LIN {X 0,Y 359.815,Z 382.386,A -85,B 0,C 180,E1 -13821.382,E2 -13821.382} C_VEL
LIN {X 0,Y 358.544,Z 382.558,A -85,B 0,C 180,E1 -13823.982,E2 -13823.982} C_VEL
LIN {X 0,Y 356.991,Z 383.681,A -85,B 0,C 180,E1 -13826.549,E2 -13826.549} C_VEL
LIN {X 0,Y 355.028,Z 386.583,A -85,B 0,C 180,E1 -13830.579,E2 -13830.579} C_VEL
LIN {X 0,Y 354.271,Z 388.561,A -85,B 0,C 180,E1 -13832.654,E2 -13832.654} C_VEL
LIN {X 0,Y 355.693,Z 391.608,A -85,B 0,C 180,E1 -13833.25,E2 -13833.25} C_VEL
LIN {X 0,Y 359.376,Z 398.785,A -85,B 0,C 180,E1 -13834.634,E2 -13834.634} C_VEL
LIN {X 0,Y 363.625,Z 409.562,A -85,B 0,C 180,E1 -13836.413,E2 -13836.413} C_VEL
LIN {X 0,Y 366.259,Z 418.959,A -85,B 0,C 180,E1 -13837.81,E2 -13837.81} C_VEL
LIN {X 0,Y 364.007,Z 432.05,A -85,B 0,C 180,E1 -13839.073,E2 -13839.073} C_VEL
LIN {X 0,Y 361.656,Z 444.882,A -85,B 0,C 180,E1 -13840.562,E2 -13840.562} C_VEL
LIN {X 0,Y 359.281,Z 457.215,A -85,B 0,C 180,E1 -13842.351,E2 -13842.351} C_VEL
LIN {X 0,Y 357.338,Z 466.693,A -85,B 0,C 180,E1 -13844.018,E2 -13844.018} C_VEL
LIN {X 0,Y 355.42,Z 475.697,A -85,B 0,C 180,E1 -13845.971,E2 -13845.971} C_VEL
LIN {X 0,Y 353.712,Z 483.022,A -85,B 0,C 180,E1 -13847.959,E2 -13847.959} C_VEL
LIN {X 0,Y 352.415,Z 488.041,A -85,B 0,C 180,E1 -13849.661,E2 -13849.661} C_VEL
LIN {X 0,Y 351.389,Z 491.946,A -85,B 0,C 180,E1 -13851.373,E2 -13851.373} C_VEL
LIN {X 0,Y 350.548,Z 494.863,A -85,B 0,C 180,E1 -13853.092,E2 -13853.092} C_VEL
LIN {X 0,Y 350.216,Z 496.262,A -85,B 0,C 180,E1 -13854.242,E2 -13854.242} C_VEL
LIN {X 0,Y 349.782,Z 497.289,A -85,B 0,C 180,E1 -13855.391,E2 -13855.391} C_VEL
LIN {X 0,Y 349.427,Z 497.902,A -85,B 0,C 180,E1 -13856.541,E2 -13856.541} C_VEL
LIN {X 0,Y 349.043,Z 498.099,A -85,B 0,C 180,E1 -13857.693,E2 -13857.693} C_VEL
LIN {X 0,Y 348.804,Z 497.883,A -85,B 0,C 180,E1 -13858.846,E2 -13858.846} C_VEL
LIN {X 0,Y 348.65,Z 497.262,A -85,B 0,C 180,E1 -13860,E2 -13860} C_VEL
LIN {X 0,Y 348.523,Z 496.239,A -85,B 0,C 180,E1 -13861.156,E2 -13861.156} C_VEL
LIN {X 0,Y 348.44,Z 494.801,A -85,B 0,C 180,E1 -13862.312,E2 -13862.312} C_VEL
LIN {X 0,Y 348.542,Z 491.806,A -85,B 0,C 180,E1 -13864.047,E2 -13864.047} C_VEL
LIN {X 0,Y 348.425,Z 487.85,A -85,B 0,C 180,E1 -13865.789,E2 -13865.789} C_VEL
LIN {X 0,Y 348.951,Z 482.756,A -85,B 0,C 180,E1 -13867.523,E2 -13867.523} C_VEL
LIN {X 0,Y 349.426,Z 475.921,A -85,B 0,C 180,E1 -13869.414,E2 -13869.414} C_VEL
LIN {X 0,Y 349.993,Z 467.529,A -85,B 0,C 180,E1 -13871.291,E2 -13871.291} C_VEL
LIN {X 0,Y 350.742,Z 458.089,A -85,B 0,C 180,E1 -13873.028,E2 -13873.028} C_VEL
LIN {X 0,Y 351.6,Z 447.694,A -85,B 0,C 180,E1 -13874.617,E2 -13874.617} C_VEL
LIN {X 0,Y 352.616,Z 435.041,A -85,B 0,C 180,E1 -13876.203,E2 -13876.203} C_VEL
LIN {X 0,Y 353.463,Z 422.474,A -85,B 0,C 180,E1 -13877.502,E2 -13877.502} C_VEL
LIN {X 0,Y 354.563,Z 408.916,A -85,B 0,C 180,E1 -13878.616,E2 -13878.616} C_VEL
LIN {X 0,Y 354.923,Z 402.075,A -85,B 0,C 180,E1 -13879.097,E2 -13879.097} C_VEL
LIN {X 0,Y 353.011,Z 392.134,A -85,B 0,C 180,E1 -13879.828,E2 -13879.828} C_VEL
LIN {X 0,Y 349.184,Z 376.619,A -85,B 0,C 180,E1 -13880.804,E2 -13880.804} C_VEL
LIN {X 0,Y 347.875,Z 371.28,A -85,B 0,C 180,E1 -13881.095,E2 -13881.095} C_VEL
LIN {X 0,Y 348.164,Z 364.382,A -85,B 0,C 180,E1 -13885.082,E2 -13885.082} C_VEL
LIN {X 0,Y 348.529,Z 357.832,A -85,B 0,C 180,E1 -13888.944,E2 -13888.944} C_VEL
LIN {X 0,Y 348.812,Z 352.473,A -85,B 0,C 180,E1 -13892.192,E2 -13892.192} C_VEL
LIN {X 0,Y 349.02,Z 347.907,A -85,B 0,C 180,E1 -13895.022,E2 -13895.022} C_VEL
LIN {X 0,Y 348.92,Z 344.539,A -85,B 0,C 180,E1 -13897.177,E2 -13897.177} C_VEL
LIN {X 0,Y 348.056,Z 338.972,A -85,B 0,C 180,E1 -13900.918,E2 -13900.918} C_VEL
LIN {X 0,Y 347.764,Z 337.48,A -85,B 0,C 180,E1 -13902.023,E2 -13902.023} C_VEL
LIN {X 0,Y 347.739,Z 337.481,A -85,B 0,C 180,E1 -13906.392,E2 -13906.392} C_VEL
LIN {X 0,Y 347.767,Z 337.702,A -85,B 0,C 180,E1 -13906.68,E2 -13906.68} C_VEL
LIN {X 0,Y 349.289,Z 344.678,A -85,B 0,C 180,E1 -13909.917,E2 -13909.917} C_VEL
LIN {X 0,Y 350.445,Z 351.066,A -85,B 0,C 180,E1 -13913.01,E2 -13913.01} C_VEL
LIN {X 0,Y 350.698,Z 355.843,A -85,B 0,C 180,E1 -13915.25,E2 -13915.25} C_VEL
LIN {X 0,Y 350.454,Z 364.261,A -85,B 0,C 180,E1 -13919.175,E2 -13919.175} C_VEL
LIN {X 0,Y 350.383,Z 371.52,A -85,B 0,C 180,E1 -13922.524,E2 -13922.524} C_VEL
LIN {X 0,Y 350.5,Z 380.256,A -85,B 0,C 180,E1 -13926.355,E2 -13926.355} C_VEL
LIN {X 0,Y 350.722,Z 387.896,A -85,B 0,C 180,E1 -13929.358,E2 -13929.358} C_VEL
LIN {X 0,Y 354.939,Z 400.483,A -85,B 0,C 180,E1 -13930.039,E2 -13930.039} C_VEL
LIN {X 0,Y 356.418,Z 406.371,A -85,B 0,C 180,E1 -13930.412,E2 -13930.412} C_VEL
LIN {X 0,Y 355.912,Z 419.475,A -85,B 0,C 180,E1 -13931.193,E2 -13931.193} C_VEL
LIN {X 0,Y 355.256,Z 430.963,A -85,B 0,C 180,E1 -13932.118,E2 -13932.118} C_VEL
LIN {X 0,Y 354.442,Z 440.978,A -85,B 0,C 180,E1 -13933.14,E2 -13933.14} C_VEL
LIN {X 0,Y 353.309,Z 452.163,A -85,B 0,C 180,E1 -13934.568,E2 -13934.568} C_VEL
LIN {X 0,Y 352.501,Z 460.293,A -85,B 0,C 180,E1 -13935.861,E2 -13935.861} C_VEL
LIN {X 0,Y 351.534,Z 467.81,A -85,B 0,C 180,E1 -13937.293,E2 -13937.293} C_VEL
LIN {X 0,Y 350.826,Z 474.233,A -85,B 0,C 180,E1 -13938.793,E2 -13938.793} C_VEL
LIN {X 0,Y 350.022,Z 480.931,A -85,B 0,C 180,E1 -13940.754,E2 -13940.754} C_VEL
LIN {X 0,Y 349.087,Z 485.6,A -85,B 0,C 180,E1 -13942.478,E2 -13942.478} C_VEL
LIN {X 0,Y 348.671,Z 489.123,A -85,B 0,C 180,E1 -13944.213,E2 -13944.213} C_VEL
LIN {X 0,Y 348.589,Z 490.915,A -85,B 0,C 180,E1 -13945.372,E2 -13945.372} C_VEL
LIN {X 0,Y 348.435,Z 492.298,A -85,B 0,C 180,E1 -13946.528,E2 -13946.528} C_VEL
LIN {X 0,Y 348.086,Z 493.891,A -85,B 0,C 180,E1 -13948.84,E2 -13948.84} C_VEL
LIN {X 0,Y 348.041,Z 494.124,A -85,B 0,C 180,E1 -13949.997,E2 -13949.997} C_VEL
LIN {X 0,Y 348.214,Z 493.353,A -85,B 0,C 180,E1 -13952.311,E2 -13952.311} C_VEL
LIN {X 0,Y 348.446,Z 492.394,A -85,B 0,C 180,E1 -13953.466,E2 -13953.466} C_VEL
LIN {X 0,Y 348.63,Z 491.062,A -85,B 0,C 180,E1 -13954.622,E2 -13954.622} C_VEL
LIN {X 0,Y 348.843,Z 488.284,A -85,B 0,C 180,E1 -13956.359,E2 -13956.359} C_VEL
LIN {X 0,Y 349.415,Z 484.462,A -85,B 0,C 180,E1 -13958.091,E2 -13958.091} C_VEL
LIN {X 0,Y 350.209,Z 479.495,A -85,B 0,C 180,E1 -13959.818,E2 -13959.818} C_VEL
LIN {X 0,Y 350.899,Z 473.265,A -85,B 0,C 180,E1 -13961.551,E2 -13961.551} C_VEL
LIN {X 0,Y 351.86,Z 465.488,A -85,B 0,C 180,E1 -13963.276,E2 -13963.276} C_VEL
LIN {X 0,Y 352.854,Z 457.514,A -85,B 0,C 180,E1 -13964.708,E2 -13964.708} C_VEL
LIN {X 0,Y 353.725,Z 448.821,A -85,B 0,C 180,E1 -13965.999,E2 -13965.999} C_VEL
LIN {X 0,Y 354.637,Z 438.034,A -85,B 0,C 180,E1 -13967.29,E2 -13967.29} C_VEL
LIN {X 0,Y 355.523,Z 426.896,A -85,B 0,C 180,E1 -13968.339,E2 -13968.339} C_VEL
LIN {X 0,Y 356.176,Z 415.355,A -85,B 0,C 180,E1 -13969.184,E2 -13969.184} C_VEL
LIN {X 0,Y 356.421,Z 405.632,A -85,B 0,C 180,E1 -13969.731,E2 -13969.731} C_VEL
LIN {X 0,Y 352.601,Z 393.285,A -85,B 0,C 180,E1 -13970.478,E2 -13970.478} C_VEL
LIN {X 0,Y 350.682,Z 387.643,A -85,B 0,C 180,E1 -13970.78,E2 -13970.78} C_VEL
LIN {X 0,Y 350.472,Z 379.042,A -85,B 0,C 180,E1 -13974.269,E2 -13974.269} C_VEL
LIN {X 0,Y 350.383,Z 370.525,A -85,B 0,C 180,E1 -13978.047,E2 -13978.047} C_VEL
LIN {X 0,Y 350.518,Z 363.233,A -85,B 0,C 180,E1 -13981.416,E2 -13981.416} C_VEL
LIN {X 0,Y 350.65,Z 358.63,A -85,B 0,C 180,E1 -13983.61,E2 -13983.61} C_VEL
LIN {X 0,Y 350.02,Z 356.826,A -85,B 0,C 180,E1 -13984.524,E2 -13984.524} C_VEL
LIN {X 0,Y 347.188,Z 354.458,A -85,B 0,C 180,E1 -13986.037,E2 -13986.037} C_VEL
LIN {X 0,Y 344.649,Z 352.626,A -85,B 0,C 180,E1 -13987.263,E2 -13987.263} C_VEL
LIN {X 0,Y 343.379,Z 350.969,A -85,B 0,C 180,E1 -13988.198,E2 -13988.198} C_VEL
LIN {X 0,Y 343.181,Z 350.325,A -85,B 0,C 180,E1 -13988.512,E2 -13988.512} C_VEL
LIN {X 0,Y 342.135,Z 345.025,A -85,B 0,C 180,E1 -13991.092,E2 -13991.092} C_VEL
LIN {X 0,Y 340.707,Z 338.358,A -85,B 0,C 180,E1 -13994.205,E2 -13994.205} C_VEL
LIN {X 0,Y 340.733,Z 338.353,A -85,B 0,C 180,E1 -13997.943,E2 -13997.943} C_VEL
LIN {X 0,Y 340.719,Z 338.355,A -85,B 0,C 180,E1 -14000.25,E2 -14000.25} C_VEL
LIN {X 0,Y 340.695,Z 338.359,A -85,B 0,C 180,E1 -14003.556,E2 -14003.556} C_VEL
LIN {X 0,Y 340.674,Z 338.361,A -85,B 0,C 180,E1 -14006.151,E2 -14006.151} C_VEL
LIN {X 0,Y 340.755,Z 338.345,A -85,B 0,C 180,E1 -14010.33,E2 -14010.33} C_VEL
LIN {X 0,Y 340.784,Z 338.341,A -85,B 0,C 180,E1 -14013.018,E2 -14013.018} C_VEL
LIN {X 0,Y 340.757,Z 338.343,A -85,B 0,C 180,E1 -14016.929,E2 -14016.929} C_VEL
LIN {X 0,Y 340.785,Z 338.341,A -85,B 0,C 180,E1 -14020.733,E2 -14020.733} C_VEL
LIN {X 0,Y 340.765,Z 338.352,A -85,B 0,C 180,E1 -14023.217,E2 -14023.217} C_VEL
LIN {X 0,Y 340.825,Z 338.338,A -85,B 0,C 180,E1 -14026.889,E2 -14026.889} C_VEL
LIN {X 0,Y 340.908,Z 338.321,A -85,B 0,C 180,E1 -14030.507,E2 -14030.507} C_VEL
LIN {X 0,Y 341.052,Z 338.314,A -85,B 0,C 180,E1 -14032.897,E2 -14032.897} C_VEL
LIN {X 0,Y 341.143,Z 338.304,A -85,B 0,C 180,E1 -14037.638,E2 -14037.638} C_VEL
LIN {X 0,Y 341.252,Z 338.281,A -85,B 0,C 180,E1 -14040,E2 -14040} C_VEL
LIN {X 0,Y 341.157,Z 338.298,A -85,B 0,C 180,E1 -14042.361,E2 -14042.361} C_VEL
LIN {X 0,Y 341.055,Z 338.313,A -85,B 0,C 180,E1 -14047.102,E2 -14047.102} C_VEL
LIN {X 0,Y 340.852,Z 338.341,A -85,B 0,C 180,E1 -14050.694,E2 -14050.694} C_VEL
LIN {X 0,Y 340.839,Z 338.344,A -85,B 0,C 180,E1 -14054.325,E2 -14054.325} C_VEL
LIN {X 0,Y 340.816,Z 338.344,A -85,B 0,C 180,E1 -14058.468,E2 -14058.468} C_VEL
LIN {X 0,Y 340.79,Z 338.346,A -85,B 0,C 180,E1 -14061.883,E2 -14061.883} C_VEL
LIN {X 0,Y 340.754,Z 338.351,A -85,B 0,C 180,E1 -14065.665,E2 -14065.665} C_VEL
LIN {X 0,Y 340.718,Z 338.356,A -85,B 0,C 180,E1 -14068.321,E2 -14068.321} C_VEL
LIN {X 0,Y 340.683,Z 338.371,A -85,B 0,C 180,E1 -14071.132,E2 -14071.132} C_VEL
LIN {X 0,Y 343.277,Z 347.352,A -85,B 0,C 180,E1 -14075.029,E2 -14075.029} C_VEL
LIN {X 0,Y 346.144,Z 357.402,A -85,B 0,C 180,E1 -14079.006,E2 -14079.006} C_VEL
LIN {X 0,Y 348.807,Z 366.887,A -85,B 0,C 180,E1 -14082.452,E2 -14082.452} C_VEL
LIN {X 0,Y 351.893,Z 377.324,A -85,B 0,C 180,E1 -14085.971,E2 -14085.971} C_VEL
LIN {X 0,Y 354.639,Z 387.6,A -85,B 0,C 180,E1 -14089.163,E2 -14089.163} C_VEL
LIN {X 0,Y 355.6,Z 391.91,A -85,B 0,C 180,E1 -14090.424,E2 -14090.424} C_VEL
LIN {X 0,Y 352.415,Z 406.455,A -85,B 0,C 180,E1 -14093.968,E2 -14093.968} C_VEL
LIN {X 0,Y 350.81,Z 414.741,A -85,B 0,C 180,E1 -14095.931,E2 -14095.931} C_VEL
LIN {X 0,Y 354.593,Z 437.489,A -85,B 0,C 180,E1 -14096.931,E2 -14096.931} C_VEL
LIN {X 0,Y 356.863,Z 453.689,A -85,B 0,C 180,E1 -14097.821,E2 -14097.821} C_VEL
LIN {X 0,Y 358.237,Z 464.384,A -85,B 0,C 180,E1 -14098.523,E2 -14098.523} C_VEL
LIN {X 0,Y 356.534,Z 480.109,A -85,B 0,C 180,E1 -14099.501,E2 -14099.501} C_VEL
LIN {X 0,Y 354.425,Z 495.314,A -85,B 0,C 180,E1 -14100.673,E2 -14100.673} C_VEL
LIN {X 0,Y 352.288,Z 509.765,A -85,B 0,C 180,E1 -14102.046,E2 -14102.046} C_VEL
LIN {X 0,Y 349.976,Z 523.578,A -85,B 0,C 180,E1 -14103.625,E2 -14103.625} C_VEL
LIN {X 0,Y 347.716,Z 536.833,A -85,B 0,C 180,E1 -14105.44,E2 -14105.44} C_VEL
LIN {X 0,Y 345.769,Z 548.209,A -85,B 0,C 180,E1 -14107.286,E2 -14107.286} C_VEL
LIN {X 0,Y 343.953,Z 559.081,A -85,B 0,C 180,E1 -14109.365,E2 -14109.365} C_VEL
LIN {X 0,Y 342.497,Z 568.353,A -85,B 0,C 180,E1 -14111.458,E2 -14111.458} C_VEL
LIN {X 0,Y 341.455,Z 576.22,A -85,B 0,C 180,E1 -14113.563,E2 -14113.563} C_VEL
LIN {X 0,Y 340.56,Z 583.613,A -85,B 0,C 180,E1 -14115.91,E2 -14115.91} C_VEL
LIN {X 0,Y 340.047,Z 589.25,A -85,B 0,C 180,E1 -14118.076,E2 -14118.076} C_VEL
LIN {X 0,Y 339.712,Z 594.263,A -85,B 0,C 180,E1 -14120.477,E2 -14120.477} C_VEL
LIN {X 0,Y 339.718,Z 598.574,A -85,B 0,C 180,E1 -14123.219,E2 -14123.219} C_VEL
LIN {X 0,Y 339.696,Z 600.784,A -85,B 0,C 180,E1 -14125.256,E2 -14125.256} C_VEL
LIN {X 0,Y 339.807,Z 601.705,A -85,B 0,C 180,E1 -14126.446,E2 -14126.446} C_VEL
LIN {X 0,Y 339.722,Z 602.725,A -85,B 0,C 180,E1 -14128.818,E2 -14128.818} C_VEL
LIN {X 0,Y 339.738,Z 602.594,A -85,B 0,C 180,E1 -14131.188,E2 -14131.188} C_VEL
LIN {X 0,Y 339.818,Z 601.433,A -85,B 0,C 180,E1 -14133.56,E2 -14133.56} C_VEL
LIN {X 0,Y 339.688,Z 599.113,A -85,B 0,C 180,E1 -14135.941,E2 -14135.941} C_VEL
LIN {X 0,Y 339.756,Z 595.701,A -85,B 0,C 180,E1 -14138.328,E2 -14138.328} C_VEL
LIN {X 0,Y 339.864,Z 591.152,A -85,B 0,C 180,E1 -14140.729,E2 -14140.729} C_VEL
LIN {X 0,Y 340.473,Z 584.037,A -85,B 0,C 180,E1 -14143.629,E2 -14143.629} C_VEL
LIN {X 0,Y 341.443,Z 575.329,A -85,B 0,C 180,E1 -14146.443,E2 -14146.443} C_VEL
LIN {X 0,Y 342.697,Z 566.272,A -85,B 0,C 180,E1 -14148.847,E2 -14148.847} C_VEL
LIN {X 0,Y 344.387,Z 555.599,A -85,B 0,C 180,E1 -14151.24,E2 -14151.24} C_VEL
LIN {X 0,Y 346.328,Z 544.712,A -85,B 0,C 180,E1 -14153.313,E2 -14153.313} C_VEL
LIN {X 0,Y 348.731,Z 532.099,A -85,B 0,C 180,E1 -14155.359,E2 -14155.359} C_VEL
LIN {X 0,Y 351.045,Z 519.623,A -85,B 0,C 180,E1 -14157.097,E2 -14157.097} C_VEL
LIN {X 0,Y 353.86,Z 504.528,A -85,B 0,C 180,E1 -14158.865,E2 -14158.865} C_VEL
LIN {X 0,Y 356.57,Z 489.422,A -85,B 0,C 180,E1 -14160.338,E2 -14160.338} C_VEL
LIN {X 0,Y 359.444,Z 472.332,A -85,B 0,C 180,E1 -14161.702,E2 -14161.702} C_VEL
LIN {X 0,Y 360.438,Z 465.571,A -85,B 0,C 180,E1 -14162.165,E2 -14162.165} C_VEL
LIN {X 0,Y 359.822,Z 450.974,A -85,B 0,C 180,E1 -14163.354,E2 -14163.354} C_VEL
LIN {X 0,Y 359.195,Z 436.999,A -85,B 0,C 180,E1 -14164.365,E2 -14164.365} C_VEL
LIN {X 0,Y 357.293,Z 423.761,A -85,B 0,C 180,E1 -14165.394,E2 -14165.394} C_VEL
LIN {X 0,Y 354.236,Z 409.339,A -85,B 0,C 180,E1 -14166.695,E2 -14166.695} C_VEL
LIN {X 0,Y 357.67,Z 399.95,A -85,B 0,C 180,E1 -14169.551,E2 -14169.551} C_VEL
LIN {X 0,Y 358.302,Z 397.75,A -85,B 0,C 180,E1 -14170.34,E2 -14170.34} C_VEL
LIN {X 0,Y 357.264,Z 393.411,A -85,B 0,C 180,E1 -14172.593,E2 -14172.593} C_VEL
LIN {X 0,Y 355.864,Z 389.527,A -85,B 0,C 180,E1 -14175.316,E2 -14175.316} C_VEL
LIN {X 0,Y 354.871,Z 387.187,A -85,B 0,C 180,E1 -14177.675,E2 -14177.675} C_VEL
LIN {X 0,Y 354.314,Z 386.23,A -85,B 0,C 180,E1 -14179.113,E2 -14179.113} C_VEL
LIN {X 0,Y 353.604,Z 385.549,A -85,B 0,C 180,E1 -14180.82,E2 -14180.82} C_VEL
LIN {X 0,Y 352.494,Z 385.363,A -85,B 0,C 180,E1 -14183.264,E2 -14183.264} C_VEL
LIN {X 0,Y 350.838,Z 386.228,A -85,B 0,C 180,E1 -14185.883,E2 -14185.883} C_VEL
LIN {X 0,Y 348.767,Z 388.633,A -85,B 0,C 180,E1 -14189.75,E2 -14189.75} C_VEL
LIN {X 0,Y 348.145,Z 389.961,A -85,B 0,C 180,E1 -14191.312,E2 -14191.312} C_VEL
LIN {X 0,Y 349.86,Z 393.47,A -85,B 0,C 180,E1 -14192.117,E2 -14192.117} C_VEL
LIN {X 0,Y 353.24,Z 400.153,A -85,B 0,C 180,E1 -14193.552,E2 -14193.552} C_VEL
LIN {X 0,Y 356.955,Z 409.105,A -85,B 0,C 180,E1 -14195.215,E2 -14195.215} C_VEL
LIN {X 0,Y 360.014,Z 419.086,A -85,B 0,C 180,E1 -14196.86,E2 -14196.86} C_VEL
LIN {X 0,Y 360.455,Z 422.118,A -85,B 0,C 180,E1 -14197.294,E2 -14197.294} C_VEL
LIN {X 0,Y 357.903,Z 435.965,A -85,B 0,C 180,E1 -14198.699,E2 -14198.699} C_VEL
LIN {X 0,Y 355.433,Z 448.064,A -85,B 0,C 180,E1 -14200.208,E2 -14200.208} C_VEL
LIN {X 0,Y 353.294,Z 458.324,A -85,B 0,C 180,E1 -14201.742,E2 -14201.742} C_VEL
LIN {X 0,Y 350.898,Z 469.156,A -85,B 0,C 180,E1 -14203.716,E2 -14203.716} C_VEL
LIN {X 0,Y 349.022,Z 477.161,A -85,B 0,C 180,E1 -14205.52,E2 -14205.52} C_VEL
LIN {X 0,Y 347.045,Z 485.046,A -85,B 0,C 180,E1 -14207.724,E2 -14207.724} C_VEL
LIN {X 0,Y 345.673,Z 489.873,A -85,B 0,C 180,E1 -14209.457,E2 -14209.457} C_VEL
LIN {X 0,Y 344.595,Z 493.651,A -85,B 0,C 180,E1 -14211.202,E2 -14211.202} C_VEL
LIN {X 0,Y 343.699,Z 496.45,A -85,B 0,C 180,E1 -14212.953,E2 -14212.953} C_VEL
LIN {X 0,Y 343.32,Z 497.77,A -85,B 0,C 180,E1 -14214.126,E2 -14214.126} C_VEL
LIN {X 0,Y 342.858,Z 498.735,A -85,B 0,C 180,E1 -14215.297,E2 -14215.297} C_VEL
LIN {X 0,Y 342.477,Z 499.268,A -85,B 0,C 180,E1 -14216.471,E2 -14216.471} C_VEL
LIN {X 0,Y 342.091,Z 499.404,A -85,B 0,C 180,E1 -14217.646,E2 -14217.646} C_VEL
LIN {X 0,Y 341.831,Z 499.129,A -85,B 0,C 180,E1 -14218.822,E2 -14218.822} C_VEL
LIN {X 0,Y 341.656,Z 498.447,A -85,B 0,C 180,E1 -14220,E2 -14220} C_VEL
LIN {X 0,Y 341.528,Z 497.365,A -85,B 0,C 180,E1 -14221.18,E2 -14221.18} C_VEL
LIN {X 0,Y 341.434,Z 495.848,A -85,B 0,C 180,E1 -14222.36,E2 -14222.36} C_VEL
LIN {X 0,Y 341.538,Z 492.764,A -85,B 0,C 180,E1 -14224.131,E2 -14224.131} C_VEL
LIN {X 0,Y 341.414,Z 488.707,A -85,B 0,C 180,E1 -14225.908,E2 -14225.908} C_VEL
LIN {X 0,Y 342.068,Z 482.532,A -85,B 0,C 180,E1 -14227.972,E2 -14227.972} C_VEL
LIN {X 0,Y 342.49,Z 475.215,A -85,B 0,C 180,E1 -14229.935,E2 -14229.935} C_VEL
LIN {X 0,Y 343.181,Z 466.57,A -85,B 0,C 180,E1 -14231.818,E2 -14231.818} C_VEL
LIN {X 0,Y 343.922,Z 456.679,A -85,B 0,C 180,E1 -14233.592,E2 -14233.592} C_VEL
LIN {X 0,Y 344.973,Z 445.734,A -85,B 0,C 180,E1 -14235.207,E2 -14235.207} C_VEL
LIN {X 0,Y 345.929,Z 433.274,A -85,B 0,C 180,E1 -14236.737,E2 -14236.737} C_VEL
LIN {X 0,Y 346.796,Z 420.672,A -85,B 0,C 180,E1 -14238.002,E2 -14238.002} C_VEL
LIN {X 0,Y 347.91,Z 407.213,A -85,B 0,C 180,E1 -14239.092,E2 -14239.092} C_VEL
LIN {X 0,Y 348.072,Z 402.371,A -85,B 0,C 180,E1 -14239.436,E2 -14239.436} C_VEL
LIN {X 0,Y 344.914,Z 388.063,A -85,B 0,C 180,E1 -14240.493,E2 -14240.493} C_VEL
LIN {X 0,Y 340.902,Z 371.644,A -85,B 0,C 180,E1 -14241.505,E2 -14241.505} C_VEL
LIN {X 0,Y 341.205,Z 364.583,A -85,B 0,C 180,E1 -14245.63,E2 -14245.63} C_VEL
LIN {X 0,Y 341.531,Z 359.093,A -85,B 0,C 180,E1 -14248.92,E2 -14248.92} C_VEL
LIN {X 0,Y 341.842,Z 353.157,A -85,B 0,C 180,E1 -14252.546,E2 -14252.546} C_VEL
LIN {X 0,Y 342.065,Z 347.941,A -85,B 0,C 180,E1 -14255.843,E2 -14255.843} C_VEL
LIN {X 0,Y 341.649,Z 343.799,A -85,B 0,C 180,E1 -14258.581,E2 -14258.581} C_VEL
LIN {X 0,Y 340.78,Z 338.747,A -85,B 0,C 180,E1 -14262.058,E2 -14262.058} C_VEL
LIN {X 0,Y 340.741,Z 338.352,A -85,B 0,C 180,E1 -14262.419,E2 -14262.419} C_VEL
LIN {X 0,Y 340.7,Z 338.505,A -85,B 0,C 180,E1 -14266.002,E2 -14266.002} C_VEL
LIN {X 0,Y 342.044,Z 344.592,A -85,B 0,C 180,E1 -14268.887,E2 -14268.887} C_VEL
LIN {X 0,Y 343.318,Z 351.214,A -85,B 0,C 180,E1 -14272.109,E2 -14272.109} C_VEL
LIN {X 0,Y 343.879,Z 355.903,A -85,B 0,C 180,E1 -14274.338,E2 -14274.338} C_VEL
LIN {X 0,Y 343.703,Z 363.478,A -85,B 0,C 180,E1 -14277.881,E2 -14277.881} C_VEL
LIN {X 0,Y 343.531,Z 372.203,A -85,B 0,C 180,E1 -14281.928,E2 -14281.928} C_VEL
LIN {X 0,Y 343.621,Z 379.609,A -85,B 0,C 180,E1 -14285.208,E2 -14285.208} C_VEL
LIN {X 0,Y 343.766,Z 387.395,A -85,B 0,C 180,E1 -14288.406,E2 -14288.406} C_VEL
LIN {X 0,Y 343.859,Z 388.871,A -85,B 0,C 180,E1 -14288.925,E2 -14288.925} C_VEL
LIN {X 0,Y 348.143,Z 401.473,A -85,B 0,C 180,E1 -14289.629,E2 -14289.629} C_VEL
LIN {X 0,Y 349.811,Z 408.243,A -85,B 0,C 180,E1 -14290.071,E2 -14290.071} C_VEL
LIN {X 0,Y 349.28,Z 420.787,A -85,B 0,C 180,E1 -14290.84,E2 -14290.84} C_VEL
LIN {X 0,Y 348.583,Z 431.988,A -85,B 0,C 180,E1 -14291.76,E2 -14291.76} C_VEL
LIN {X 0,Y 347.732,Z 442.046,A -85,B 0,C 180,E1 -14292.805,E2 -14292.805} C_VEL
LIN {X 0,Y 346.547,Z 453.235,A -85,B 0,C 180,E1 -14294.259,E2 -14294.259} C_VEL
LIN {X 0,Y 345.7,Z 461.367,A -85,B 0,C 180,E1 -14295.577,E2 -14295.577} C_VEL
LIN {X 0,Y 344.701,Z 468.883,A -85,B 0,C 180,E1 -14297.037,E2 -14297.037} C_VEL
LIN {X 0,Y 343.955,Z 475.257,A -85,B 0,C 180,E1 -14298.552,E2 -14298.552} C_VEL
LIN {X 0,Y 343.104,Z 482.006,A -85,B 0,C 180,E1 -14300.566,E2 -14300.566} C_VEL
LIN {X 0,Y 342.131,Z 486.677,A -85,B 0,C 180,E1 -14302.324,E2 -14302.324} C_VEL
LIN {X 0,Y 341.691,Z 490.2,A -85,B 0,C 180,E1 -14304.094,E2 -14304.094} C_VEL
LIN {X 0,Y 341.611,Z 491.99,A -85,B 0,C 180,E1 -14305.277,E2 -14305.277} C_VEL
LIN {X 0,Y 341.432,Z 493.375,A -85,B 0,C 180,E1 -14306.457,E2 -14306.457} C_VEL
LIN {X 0,Y 341.07,Z 494.968,A -85,B 0,C 180,E1 -14308.816,E2 -14308.816} C_VEL
LIN {X 0,Y 341.046,Z 495.197,A -85,B 0,C 180,E1 -14309.997,E2 -14309.997} C_VEL
LIN {X 0,Y 341.203,Z 494.43,A -85,B 0,C 180,E1 -14312.358,E2 -14312.358} C_VEL
LIN {X 0,Y 341.443,Z 493.47,A -85,B 0,C 180,E1 -14313.537,E2 -14313.537} C_VEL
LIN {X 0,Y 341.645,Z 492.136,A -85,B 0,C 180,E1 -14314.717,E2 -14314.717} C_VEL
LIN {X 0,Y 341.867,Z 489.36,A -85,B 0,C 180,E1 -14316.489,E2 -14316.489} C_VEL
LIN {X 0,Y 342.469,Z 485.536,A -85,B 0,C 180,E1 -14318.256,E2 -14318.256} C_VEL
LIN {X 0,Y 343.301,Z 480.567,A -85,B 0,C 180,E1 -14320.018,E2 -14320.018} C_VEL
LIN {X 0,Y 344.023,Z 474.337,A -85,B 0,C 180,E1 -14321.785,E2 -14321.785} C_VEL
LIN {X 0,Y 345.033,Z 466.558,A -85,B 0,C 180,E1 -14323.544,E2 -14323.544} C_VEL
LIN {X 0,Y 346.069,Z 458.581,A -85,B 0,C 180,E1 -14325.003,E2 -14325.003} C_VEL
LIN {X 0,Y 346.981,Z 449.885,A -85,B 0,C 180,E1 -14326.319,E2 -14326.319} C_VEL
LIN {X 0,Y 347.94,Z 439.091,A -85,B 0,C 180,E1 -14327.634,E2 -14327.634} C_VEL
LIN {X 0,Y 348.88,Z 427.943,A -85,B 0,C 180,E1 -14328.701,E2 -14328.701} C_VEL
LIN {X 0,Y 349.566,Z 415.79,A -85,B 0,C 180,E1 -14329.6,E2 -14329.6} C_VEL
LIN {X 0,Y 349.744,Z 407.09,A -85,B 0,C 180,E1 -14330.101,E2 -14330.101} C_VEL
LIN {X 0,Y 346.163,Z 395.379,A -85,B 0,C 180,E1 -14330.843,E2 -14330.843} C_VEL
LIN {X 0,Y 343.839,Z 388.706,A -85,B 0,C 180,E1 -14331.19,E2 -14331.19} C_VEL
LIN {X 0,Y 343.641,Z 381.411,A -85,B 0,C 180,E1 -14334.14,E2 -14334.14} C_VEL
LIN {X 0,Y 343.568,Z 374.026,A -85,B 0,C 180,E1 -14337.4,E2 -14337.4} C_VEL
LIN {X 0,Y 343.658,Z 366.58,A -85,B 0,C 180,E1 -14340.803,E2 -14340.803} C_VEL
LIN {X 0,Y 343.919,Z 357.864,A -85,B 0,C 180,E1 -14344.898,E2 -14344.898} C_VEL
LIN {X 0,Y 343.616,Z 353.19,A -85,B 0,C 180,E1 -14347.091,E2 -14347.091} C_VEL
LIN {X 0,Y 343.181,Z 350.325,A -85,B 0,C 180,E1 -14348.512,E2 -14348.512} C_VEL
LIN {X 0,Y 342.163,Z 348.602,A -85,B 0,C 180,E1 -14349.439,E2 -14349.439} C_VEL
LIN {X 0,Y 338.792,Z 346.418,A -85,B 0,C 180,E1 -14350.963,E2 -14350.963} C_VEL
LIN {X 0,Y 335.944,Z 344.578,A -85,B 0,C 180,E1 -14352.197,E2 -14352.197} C_VEL
LIN {X 0,Y 334.527,Z 342.849,A -85,B 0,C 180,E1 -14353.144,E2 -14353.144} C_VEL
LIN {X 0,Y 334.299,Z 342.177,A -85,B 0,C 180,E1 -14353.462,E2 -14353.462} C_VEL
LIN {X 0,Y 333.66,Z 339.236,A -85,B 0,C 180,E1 -14354.856,E2 -14354.856} C_VEL
LIN {X 0,Y 333.679,Z 339.232,A -85,B 0,C 180,E1 -14357.624,E2 -14357.624} C_VEL
LIN {X 0,Y 333.668,Z 339.235,A -85,B 0,C 180,E1 -14361.193,E2 -14361.193} C_VEL
LIN {X 0,Y 333.668,Z 339.234,A -85,B 0,C 180,E1 -14365.223,E2 -14365.223} C_VEL
LIN {X 0,Y 333.679,Z 339.228,A -85,B 0,C 180,E1 -14369.635,E2 -14369.635} C_VEL
LIN {X 0,Y 333.723,Z 339.227,A -85,B 0,C 180,E1 -14372.399,E2 -14372.399} C_VEL
LIN {X 0,Y 333.741,Z 339.226,A -85,B 0,C 180,E1 -14375.091,E2 -14375.091} C_VEL
LIN {X 0,Y 333.703,Z 339.23,A -85,B 0,C 180,E1 -14379.02,E2 -14379.02} C_VEL
LIN {X 0,Y 333.774,Z 339.213,A -85,B 0,C 180,E1 -14381.588,E2 -14381.588} C_VEL
LIN {X 0,Y 333.786,Z 339.207,A -85,B 0,C 180,E1 -14385.575,E2 -14385.575} C_VEL
LIN {X 0,Y 333.817,Z 339.213,A -85,B 0,C 180,E1 -14389.077,E2 -14389.077} C_VEL
LIN {X 0,Y 334.002,Z 339.192,A -85,B 0,C 180,E1 -14392.747,E2 -14392.747} C_VEL
LIN {X 0,Y 333.785,Z 339.208,A -85,B 0,C 180,E1 -14395.168,E2 -14395.168} C_VEL
LIN {X 0,Y 334.08,Z 339.184,A -85,B 0,C 180,E1 -14397.588,E2 -14397.588} C_VEL
LIN {X 0,Y 334.204,Z 339.158,A -85,B 0,C 180,E1 -14400,E2 -14400} C_VEL
LIN {X 0,Y 334.119,Z 339.175,A -85,B 0,C 180,E1 -14402.411,E2 -14402.411} C_VEL
LIN {X 0,Y 334.004,Z 339.192,A -85,B 0,C 180,E1 -14407.252,E2 -14407.252} C_VEL
LIN {X 0,Y 333.814,Z 339.217,A -85,B 0,C 180,E1 -14410.922,E2 -14410.922} C_VEL
LIN {X 0,Y 333.785,Z 339.22,A -85,B 0,C 180,E1 -14414.635,E2 -14414.635} C_VEL
LIN {X 0,Y 333.775,Z 339.221,A -85,B 0,C 180,E1 -14418.657,E2 -14418.657} C_VEL
LIN {X 0,Y 333.726,Z 339.227,A -85,B 0,C 180,E1 -14422.275,E2 -14422.275} C_VEL
LIN {X 0,Y 333.715,Z 339.227,A -85,B 0,C 180,E1 -14426.247,E2 -14426.247} C_VEL
LIN {X 0,Y 333.686,Z 339.309,A -85,B 0,C 180,E1 -14430.177,E2 -14430.177} C_VEL
LIN {X 0,Y 336.314,Z 348.652,A -85,B 0,C 180,E1 -14434.348,E2 -14434.348} C_VEL
LIN {X 0,Y 338.865,Z 357.571,A -85,B 0,C 180,E1 -14437.997,E2 -14437.997} C_VEL
LIN {X 0,Y 341.588,Z 367.203,A -85,B 0,C 180,E1 -14441.624,E2 -14441.624} C_VEL
LIN {X 0,Y 344.832,Z 378.406,A -85,B 0,C 180,E1 -14445.506,E2 -14445.506} C_VEL
LIN {X 0,Y 347.626,Z 388.765,A -85,B 0,C 180,E1 -14448.808,E2 -14448.808} C_VEL
LIN {X 0,Y 348.757,Z 393.382,A -85,B 0,C 180,E1 -14450.198,E2 -14450.198} C_VEL
LIN {X 0,Y 345.745,Z 406.685,A -85,B 0,C 180,E1 -14453.523,E2 -14453.523} C_VEL
LIN {X 0,Y 344.169,Z 414.44,A -85,B 0,C 180,E1 -14455.403,E2 -14455.403} C_VEL
LIN {X 0,Y 347.786,Z 437.013,A -85,B 0,C 180,E1 -14456.413,E2 -14456.413} C_VEL
LIN {X 0,Y 350.147,Z 453.357,A -85,B 0,C 180,E1 -14457.338,E2 -14457.338} C_VEL
LIN {X 0,Y 351.555,Z 465.355,A -85,B 0,C 180,E1 -14458.142,E2 -14458.142} C_VEL
LIN {X 0,Y 349.74,Z 481.28,A -85,B 0,C 180,E1 -14459.179,E2 -14459.179} C_VEL
LIN {X 0,Y 347.518,Z 496.549,A -85,B 0,C 180,E1 -14460.412,E2 -14460.412} C_VEL
LIN {X 0,Y 345.406,Z 510.339,A -85,B 0,C 180,E1 -14461.77,E2 -14461.77} C_VEL
LIN {X 0,Y 343.051,Z 523.95,A -85,B 0,C 180,E1 -14463.379,E2 -14463.379} C_VEL
LIN {X 0,Y 340.852,Z 536.317,A -85,B 0,C 180,E1 -14465.125,E2 -14465.125} C_VEL
LIN {X 0,Y 338.753,Z 548.222,A -85,B 0,C 180,E1 -14467.111,E2 -14467.111} C_VEL
LIN {X 0,Y 336.907,Z 558.959,A -85,B 0,C 180,E1 -14469.233,E2 -14469.233} C_VEL
LIN {X 0,Y 335.421,Z 568.147,A -85,B 0,C 180,E1 -14471.369,E2 -14471.369} C_VEL
LIN {X 0,Y 334.377,Z 575.916,A -85,B 0,C 180,E1 -14473.52,E2 -14473.52} C_VEL
LIN {X 0,Y 333.467,Z 583.394,A -85,B 0,C 180,E1 -14475.99,E2 -14475.99} C_VEL
LIN {X 0,Y 332.912,Z 589.436,A -85,B 0,C 180,E1 -14478.434,E2 -14478.434} C_VEL
LIN {X 0,Y 332.66,Z 594.205,A -85,B 0,C 180,E1 -14480.886,E2 -14480.886} C_VEL
LIN {X 0,Y 332.667,Z 597.593,A -85,B 0,C 180,E1 -14483.18,E2 -14483.18} C_VEL
LIN {X 0,Y 332.664,Z 599.695,A -85,B 0,C 180,E1 -14485.155,E2 -14485.155} C_VEL
LIN {X 0,Y 332.778,Z 600.635,A -85,B 0,C 180,E1 -14486.37,E2 -14486.37} C_VEL
LIN {X 0,Y 332.697,Z 601.68,A -85,B 0,C 180,E1 -14488.793,E2 -14488.793} C_VEL
LIN {X 0,Y 332.712,Z 601.554,A -85,B 0,C 180,E1 -14491.213,E2 -14491.213} C_VEL
LIN {X 0,Y 332.791,Z 600.411,A -85,B 0,C 180,E1 -14493.635,E2 -14493.635} C_VEL
LIN {X 0,Y 332.648,Z 598.085,A -85,B 0,C 180,E1 -14496.067,E2 -14496.067} C_VEL
LIN {X 0,Y 332.708,Z 594.681,A -85,B 0,C 180,E1 -14498.506,E2 -14498.506} C_VEL
LIN {X 0,Y 332.819,Z 590.129,A -85,B 0,C 180,E1 -14500.958,E2 -14500.958} C_VEL
LIN {X 0,Y 333.329,Z 584.346,A -85,B 0,C 180,E1 -14503.413,E2 -14503.413} C_VEL
LIN {X 0,Y 334.072,Z 577.322,A -85,B 0,C 180,E1 -14505.874,E2 -14505.874} C_VEL
LIN {X 0,Y 335.248,Z 568.938,A -85,B 0,C 180,E1 -14508.33,E2 -14508.33} C_VEL
LIN {X 0,Y 337.118,Z 557.608,A -85,B 0,C 180,E1 -14511.079,E2 -14511.079} C_VEL
LIN {X 0,Y 339.354,Z 545.653,A -85,B 0,C 180,E1 -14513.497,E2 -14513.497} C_VEL
LIN {X 0,Y 341.81,Z 533.424,A -85,B 0,C 180,E1 -14515.583,E2 -14515.583} C_VEL
LIN {X 0,Y 344.406,Z 520.251,A -85,B 0,C 180,E1 -14517.499,E2 -14517.499} C_VEL
LIN {X 0,Y 347.242,Z 506.142,A -85,B 0,C 180,E1 -14519.232,E2 -14519.232} C_VEL
LIN {X 0,Y 350.161,Z 491.064,A -85,B 0,C 180,E1 -14520.787,E2 -14520.787} C_VEL
LIN {X 0,Y 353.171,Z 474.803,A -85,B 0,C 180,E1 -14522.165,E2 -14522.165} C_VEL
LIN {X 0,Y 354.367,Z 468.093,A -85,B 0,C 180,E1 -14522.651,E2 -14522.651} C_VEL
LIN {X 0,Y 354.155,Z 452.147,A -85,B 0,C 180,E1 -14524.017,E2 -14524.017} C_VEL
LIN {X 0,Y 353.809,Z 439.473,A -85,B 0,C 180,E1 -14524.994,E2 -14524.994} C_VEL
LIN {X 0,Y 352.405,Z 427.065,A -85,B 0,C 180,E1 -14526.031,E2 -14526.031} C_VEL
LIN {X 0,Y 349.554,Z 412.659,A -85,B 0,C 180,E1 -14527.413,E2 -14527.413} C_VEL
LIN {X 0,Y 348.724,Z 408.452,A -85,B 0,C 180,E1 -14527.87,E2 -14527.87} C_VEL
LIN {X 0,Y 351.696,Z 400.851,A -85,B 0,C 180,E1 -14530.337,E2 -14530.337} C_VEL
LIN {X 0,Y 351.476,Z 398.832,A -85,B 0,C 180,E1 -14531.292,E2 -14531.292} C_VEL
LIN {X 0,Y 350.273,Z 394.674,A -85,B 0,C 180,E1 -14533.755,E2 -14533.755} C_VEL
LIN {X 0,Y 348.848,Z 391.086,A -85,B 0,C 180,E1 -14536.767,E2 -14536.767} C_VEL
LIN {X 0,Y 348.214,Z 389.833,A -85,B 0,C 180,E1 -14538.314,E2 -14538.314} C_VEL
LIN {X 0,Y 347.042,Z 388.532,A -85,B 0,C 180,E1 -14541.114,E2 -14541.114} C_VEL
LIN {X 0,Y 346.382,Z 388.352,A -85,B 0,C 180,E1 -14542.506,E2 -14542.506} C_VEL
LIN {X 0,Y 344.724,Z 388.893,A -85,B 0,C 180,E1 -14545.191,E2 -14545.191} C_VEL
LIN {X 0,Y 342.475,Z 390.965,A -85,B 0,C 180,E1 -14549.135,E2 -14549.135} C_VEL
LIN {X 0,Y 342.201,Z 391.42,A -85,B 0,C 180,E1 -14549.773,E2 -14549.773} C_VEL
LIN {X 0,Y 343.652,Z 394.678,A -85,B 0,C 180,E1 -14550.606,E2 -14550.606} C_VEL
LIN {X 0,Y 344.865,Z 396.862,A -85,B 0,C 180,E1 -14551.202,E2 -14551.202} C_VEL
LIN {X 0,Y 348.978,Z 405.376,A -85,B 0,C 180,E1 -14553.186,E2 -14553.186} C_VEL
LIN {X 0,Y 352.166,Z 413.896,A -85,B 0,C 180,E1 -14554.859,E2 -14554.859} C_VEL
LIN {X 0,Y 354.751,Z 423.297,A -85,B 0,C 180,E1 -14556.496,E2 -14556.496} C_VEL
LIN {X 0,Y 354.898,Z 424.469,A -85,B 0,C 180,E1 -14556.669,E2 -14556.669} C_VEL
LIN {X 0,Y 352.319,Z 437.466,A -85,B 0,C 180,E1 -14558.037,E2 -14558.037} C_VEL
LIN {X 0,Y 349.463,Z 450.43,A -85,B 0,C 180,E1 -14559.702,E2 -14559.702} C_VEL
LIN {X 0,Y 347.01,Z 461.221,A -85,B 0,C 180,E1 -14561.399,E2 -14561.399} C_VEL
LIN {X 0,Y 344.815,Z 470.323,A -85,B 0,C 180,E1 -14563.116,E2 -14563.116} C_VEL
LIN {X 0,Y 342.583,Z 479.068,A -85,B 0,C 180,E1 -14565.142,E2 -14565.142} C_VEL
LIN {X 0,Y 340.919,Z 485.215,A -85,B 0,C 180,E1 -14566.894,E2 -14566.894} C_VEL
LIN {X 0,Y 339.39,Z 490.272,A -85,B 0,C 180,E1 -14568.655,E2 -14568.655} C_VEL
LIN {X 0,Y 338.109,Z 494.272,A -85,B 0,C 180,E1 -14570.428,E2 -14570.428} C_VEL
LIN {X 0,Y 336.861,Z 498.04,A -85,B 0,C 180,E1 -14572.809,E2 -14572.809} C_VEL
LIN {X 0,Y 336.435,Z 499.308,A -85,B 0,C 180,E1 -14574.005,E2 -14574.005} C_VEL
LIN {X 0,Y 335.945,Z 500.179,A -85,B 0,C 180,E1 -14575.2,E2 -14575.2} C_VEL
LIN {X 0,Y 335.538,Z 500.626,A -85,B 0,C 180,E1 -14576.398,E2 -14576.398} C_VEL
LIN {X 0,Y 335.13,Z 500.7,A -85,B 0,C 180,E1 -14577.597,E2 -14577.597} C_VEL
LIN {X 0,Y 334.853,Z 500.367,A -85,B 0,C 180,E1 -14578.798,E2 -14578.798} C_VEL
LIN {X 0,Y 334.658,Z 499.627,A -85,B 0,C 180,E1 -14580,E2 -14580} C_VEL
LIN {X 0,Y 334.53,Z 498.471,A -85,B 0,C 180,E1 -14581.204,E2 -14581.204} C_VEL
LIN {X 0,Y 334.445,Z 495.933,A -85,B 0,C 180,E1 -14583.012,E2 -14583.012} C_VEL
LIN {X 0,Y 334.463,Z 492.416,A -85,B 0,C 180,E1 -14584.822,E2 -14584.822} C_VEL
LIN {X 0,Y 334.626,Z 487.874,A -85,B 0,C 180,E1 -14586.634,E2 -14586.634} C_VEL
LIN {X 0,Y 335.182,Z 482.2,A -85,B 0,C 180,E1 -14588.441,E2 -14588.441} C_VEL
LIN {X 0,Y 335.654,Z 474.467,A -85,B 0,C 180,E1 -14590.46,E2 -14590.46} C_VEL
LIN {X 0,Y 336.379,Z 465.45,A -85,B 0,C 180,E1 -14592.366,E2 -14592.366} C_VEL
LIN {X 0,Y 337.161,Z 455.127,A -85,B 0,C 180,E1 -14594.178,E2 -14594.178} C_VEL
LIN {X 0,Y 338.295,Z 443.666,A -85,B 0,C 180,E1 -14595.824,E2 -14595.824} C_VEL
LIN {X 0,Y 339.346,Z 430.383,A -85,B 0,C 180,E1 -14597.394,E2 -14597.394} C_VEL
LIN {X 0,Y 340.165,Z 418.85,A -85,B 0,C 180,E1 -14598.522,E2 -14598.522} C_VEL
LIN {X 0,Y 341.291,Z 404.169,A -85,B 0,C 180,E1 -14599.67,E2 -14599.67} C_VEL
LIN {X 0,Y 338.26,Z 389.848,A -85,B 0,C 180,E1 -14600.773,E2 -14600.773} C_VEL
LIN {X 0,Y 334.135,Z 373.283,A -85,B 0,C 180,E1 -14601.811,E2 -14601.811} C_VEL
LIN {X 0,Y 333.909,Z 372.058,A -85,B 0,C 180,E1 -14601.898,E2 -14601.898} C_VEL
LIN {X 0,Y 334.136,Z 366.38,A -85,B 0,C 180,E1 -14605.249,E2 -14605.249} C_VEL
LIN {X 0,Y 334.525,Z 360.348,A -85,B 0,C 180,E1 -14608.895,E2 -14608.895} C_VEL
LIN {X 0,Y 334.887,Z 353.604,A -85,B 0,C 180,E1 -14613.069,E2 -14613.069} C_VEL
LIN {X 0,Y 335.099,Z 349.078,A -85,B 0,C 180,E1 -14615.962,E2 -14615.962} C_VEL
LIN {X 0,Y 334.768,Z 345.702,A -85,B 0,C 180,E1 -14618.231,E2 -14618.231} C_VEL
LIN {X 0,Y 333.972,Z 340.954,A -85,B 0,C 180,E1 -14621.519,E2 -14621.519} C_VEL
LIN {X 0,Y 333.694,Z 339.229,A -85,B 0,C 180,E1 -14622.812,E2 -14622.812} C_VEL
LIN {X 0,Y 333.652,Z 339.325,A -85,B 0,C 180,E1 -14625.337,E2 -14625.337} C_VEL
LIN {X 0,Y 335.078,Z 345.538,A -85,B 0,C 180,E1 -14628.277,E2 -14628.277} C_VEL
LIN {X 0,Y 336.49,Z 353.027,A -85,B 0,C 180,E1 -14631.93,E2 -14631.93} C_VEL
LIN {X 0,Y 337.058,Z 358.132,A -85,B 0,C 180,E1 -14634.41,E2 -14634.41} C_VEL
LIN {X 0,Y 336.867,Z 365.452,A -85,B 0,C 180,E1 -14637.857,E2 -14637.857} C_VEL
LIN {X 0,Y 336.707,Z 374.413,A -85,B 0,C 180,E1 -14641.987,E2 -14641.987} C_VEL
LIN {X 0,Y 336.812,Z 382.009,A -85,B 0,C 180,E1 -14645.332,E2 -14645.332} C_VEL
LIN {X 0,Y 336.966,Z 389.687,A -85,B 0,C 180,E1 -14648.456,E2 -14648.456} C_VEL
LIN {X 0,Y 341.423,Z 402.786,A -85,B 0,C 180,E1 -14649.221,E2 -14649.221} C_VEL
LIN {X 0,Y 343.205,Z 409.705,A -85,B 0,C 180,E1 -14649.694,E2 -14649.694} C_VEL
LIN {X 0,Y 342.657,Z 422.064,A -85,B 0,C 180,E1 -14650.471,E2 -14650.471} C_VEL
LIN {X 0,Y 341.923,Z 433.013,A -85,B 0,C 180,E1 -14651.388,E2 -14651.388} C_VEL
LIN {X 0,Y 341.046,Z 443.112,A -85,B 0,C 180,E1 -14652.457,E2 -14652.457} C_VEL
LIN {X 0,Y 339.796,Z 454.306,A -85,B 0,C 180,E1 -14653.938,E2 -14653.938} C_VEL
LIN {X 0,Y 338.913,Z 462.439,A -85,B 0,C 180,E1 -14655.281,E2 -14655.281} C_VEL
LIN {X 0,Y 337.872,Z 469.957,A -85,B 0,C 180,E1 -14656.77,E2 -14656.77} C_VEL
LIN {X 0,Y 337.085,Z 476.29,A -85,B 0,C 180,E1 -14658.304,E2 -14658.304} C_VEL
LIN {X 0,Y 336.188,Z 483.082,A -85,B 0,C 180,E1 -14660.37,E2 -14660.37} C_VEL
LIN {X 0,Y 335.178,Z 487.754,A -85,B 0,C 180,E1 -14662.164,E2 -14662.164} C_VEL
LIN {X 0,Y 334.712,Z 491.277,A -85,B 0,C 180,E1 -14663.971,E2 -14663.971} C_VEL
LIN {X 0,Y 334.63,Z 493.066,A -85,B 0,C 180,E1 -14665.178,E2 -14665.178} C_VEL
LIN {X 0,Y 334.429,Z 494.452,A -85,B 0,C 180,E1 -14666.383,E2 -14666.383} C_VEL
LIN {X 0,Y 334.055,Z 496.045,A -85,B 0,C 180,E1 -14668.792,E2 -14668.792} C_VEL
LIN {X 0,Y 334.048,Z 496.271,A -85,B 0,C 180,E1 -14669.997,E2 -14669.997} C_VEL
LIN {X 0,Y 334.192,Z 495.506,A -85,B 0,C 180,E1 -14672.408,E2 -14672.408} C_VEL
LIN {X 0,Y 334.44,Z 494.546,A -85,B 0,C 180,E1 -14673.611,E2 -14673.611} C_VEL
LIN {X 0,Y 334.659,Z 493.211,A -85,B 0,C 180,E1 -14674.816,E2 -14674.816} C_VEL
LIN {X 0,Y 334.892,Z 490.435,A -85,B 0,C 180,E1 -14676.625,E2 -14676.625} C_VEL
LIN {X 0,Y 335.525,Z 486.611,A -85,B 0,C 180,E1 -14678.428,E2 -14678.428} C_VEL
LIN {X 0,Y 336.397,Z 481.639,A -85,B 0,C 180,E1 -14680.226,E2 -14680.226} C_VEL
LIN {X 0,Y 337.177,Z 475.405,A -85,B 0,C 180,E1 -14682.027,E2 -14682.027} C_VEL
LIN {X 0,Y 338.213,Z 467.627,A -85,B 0,C 180,E1 -14683.822,E2 -14683.822} C_VEL
LIN {X 0,Y 339.292,Z 459.648,A -85,B 0,C 180,E1 -14685.31,E2 -14685.31} C_VEL
LIN {X 0,Y 340.249,Z 450.948,A -85,B 0,C 180,E1 -14686.651,E2 -14686.651} C_VEL
LIN {X 0,Y 341.256,Z 440.148,A -85,B 0,C 180,E1 -14687.991,E2 -14687.991} C_VEL
LIN {X 0,Y 342.238,Z 428.951,A -85,B 0,C 180,E1 -14689.082,E2 -14689.082} C_VEL
LIN {X 0,Y 342.939,Z 417.351,A -85,B 0,C 180,E1 -14689.961,E2 -14689.961} C_VEL
LIN {X 0,Y 343.184,Z 408.983,A -85,B 0,C 180,E1 -14690.454,E2 -14690.454} C_VEL
LIN {X 0,Y 339.878,Z 397.974,A -85,B 0,C 180,E1 -14691.186,E2 -14691.186} C_VEL
LIN {X 0,Y 337.016,Z 389.654,A -85,B 0,C 180,E1 -14691.672,E2 -14691.672} C_VEL
LIN {X 0,Y 336.811,Z 380.776,A -85,B 0,C 180,E1 -14695.322,E2 -14695.322} C_VEL
LIN {X 0,Y 336.793,Z 371.697,A -85,B 0,C 180,E1 -14699.361,E2 -14699.361} C_VEL
LIN {X 0,Y 336.967,Z 363.003,A -85,B 0,C 180,E1 -14703.46,E2 -14703.46} C_VEL
LIN {X 0,Y 337.065,Z 358.238,A -85,B 0,C 180,E1 -14705.715,E2 -14705.715} C_VEL
LIN {X 0,Y 336.524,Z 353.286,A -85,B 0,C 180,E1 -14708.068,E2 -14708.068} C_VEL
LIN {X 0,Y 335.419,Z 347.348,A -85,B 0,C 180,E1 -14711.035,E2 -14711.035} C_VEL
LIN {X 0,Y 334.299,Z 342.177,A -85,B 0,C 180,E1 -14713.462,E2 -14713.462} C_VEL
LIN {X 0,Y 333.357,Z 341.056,A -85,B 0,C 180,E1 -14714.099,E2 -14714.099} C_VEL
LIN {X 0,Y 330.243,Z 340.211,A -85,B 0,C 180,E1 -14715.125,E2 -14715.125} C_VEL
LIN {X 0,Y 327.283,Z 340.094,A -85,B 0,C 180,E1 -14716.193,E2 -14716.193} C_VEL
LIN {X 0,Y 326.608,Z 340.116,A -85,B 0,C 180,E1 -14716.888,E2 -14716.888} C_VEL
LIN {X 0,Y 326.63,Z 340.113,A -85,B 0,C 180,E1 -14720.763,E2 -14720.763} C_VEL
LIN {X 0,Y 326.596,Z 340.112,A -85,B 0,C 180,E1 -14724.478,E2 -14724.478} C_VEL
LIN {X 0,Y 326.59,Z 340.113,A -85,B 0,C 180,E1 -14727.453,E2 -14727.453} C_VEL
LIN {X 0,Y 326.641,Z 340.103,A -85,B 0,C 180,E1 -14730.338,E2 -14730.338} C_VEL
LIN {X 0,Y 326.674,Z 340.103,A -85,B 0,C 180,E1 -14734.514,E2 -14734.514} C_VEL
LIN {X 0,Y 326.655,Z 340.108,A -85,B 0,C 180,E1 -14738.545,E2 -14738.545} C_VEL
LIN {X 0,Y 326.723,Z 340.09,A -85,B 0,C 180,E1 -14741.176,E2 -14741.176} C_VEL
LIN {X 0,Y 326.741,Z 340.085,A -85,B 0,C 180,E1 -14745.432,E2 -14745.432} C_VEL
LIN {X 0,Y 326.752,Z 340.094,A -85,B 0,C 180,E1 -14748.838,E2 -14748.838} C_VEL
LIN {X 0,Y 326.956,Z 340.07,A -85,B 0,C 180,E1 -14752.589,E2 -14752.589} C_VEL
LIN {X 0,Y 326.752,Z 340.085,A -85,B 0,C 180,E1 -14755.064,E2 -14755.064} C_VEL
LIN {X 0,Y 327.021,Z 340.063,A -85,B 0,C 180,E1 -14757.536,E2 -14757.536} C_VEL
LIN {X 0,Y 327.156,Z 340.036,A -85,B 0,C 180,E1 -14760,E2 -14760} C_VEL
LIN {X 0,Y 327.056,Z 340.055,A -85,B 0,C 180,E1 -14762.463,E2 -14762.463} C_VEL
LIN {X 0,Y 326.977,Z 340.068,A -85,B 0,C 180,E1 -14766.169,E2 -14766.169} C_VEL
LIN {X 0,Y 326.891,Z 340.079,A -85,B 0,C 180,E1 -14768.655,E2 -14768.655} C_VEL
LIN {X 0,Y 326.715,Z 340.103,A -85,B 0,C 180,E1 -14772.422,E2 -14772.422} C_VEL
LIN {X 0,Y 326.731,Z 340.098,A -85,B 0,C 180,E1 -14774.958,E2 -14774.958} C_VEL
LIN {X 0,Y 326.741,Z 340.098,A -85,B 0,C 180,E1 -14778.855,E2 -14778.855} C_VEL
LIN {X 0,Y 326.675,Z 340.106,A -85,B 0,C 180,E1 -14782.783,E2 -14782.783} C_VEL
LIN {X 0,Y 326.663,Z 340.106,A -85,B 0,C 180,E1 -14786.859,E2 -14786.859} C_VEL
LIN {X 0,Y 326.69,Z 340.267,A -85,B 0,C 180,E1 -14789.213,E2 -14789.213} C_VEL
LIN {X 0,Y 329.131,Z 349.139,A -85,B 0,C 180,E1 -14793.307,E2 -14793.307} C_VEL
LIN {X 0,Y 331.238,Z 356.498,A -85,B 0,C 180,E1 -14796.447,E2 -14796.447} C_VEL
LIN {X 0,Y 333.757,Z 365.367,A -85,B 0,C 180,E1 -14799.959,E2 -14799.959} C_VEL
LIN {X 0,Y 337.131,Z 377.243,A -85,B 0,C 180,E1 -14804.27,E2 -14804.27} C_VEL
LIN {X 0,Y 339.678,Z 386.43,A -85,B 0,C 180,E1 -14807.342,E2 -14807.342} C_VEL
LIN {X 0,Y 341.904,Z 395.008,A -85,B 0,C 180,E1 -14810.025,E2 -14810.025} C_VEL
LIN {X 0,Y 338.539,Z 409.318,A -85,B 0,C 180,E1 -14813.677,E2 -14813.677} C_VEL
LIN {X 0,Y 337.514,Z 414.02,A -85,B 0,C 180,E1 -14814.856,E2 -14814.856} C_VEL
LIN {X 0,Y 341.075,Z 436.73,A -85,B 0,C 180,E1 -14815.897,E2 -14815.897} C_VEL
LIN {X 0,Y 343.208,Z 451.736,A -85,B 0,C 180,E1 -14816.755,E2 -14816.755} C_VEL
LIN {X 0,Y 344.864,Z 466.284,A -85,B 0,C 180,E1 -14817.759,E2 -14817.759} C_VEL
LIN {X 0,Y 342.939,Z 482.216,A -85,B 0,C 180,E1 -14818.842,E2 -14818.842} C_VEL
LIN {X 0,Y 340.541,Z 497.88,A -85,B 0,C 180,E1 -14820.164,E2 -14820.164} C_VEL
LIN {X 0,Y 338.343,Z 512.027,A -85,B 0,C 180,E1 -14821.635,E2 -14821.635} C_VEL
LIN {X 0,Y 335.915,Z 525.275,A -85,B 0,C 180,E1 -14823.272,E2 -14823.272} C_VEL
LIN {X 0,Y 333.643,Z 537.624,A -85,B 0,C 180,E1 -14825.088,E2 -14825.088} C_VEL
LIN {X 0,Y 331.457,Z 549.846,A -85,B 0,C 180,E1 -14827.238,E2 -14827.238} C_VEL
LIN {X 0,Y 329.555,Z 560.457,A -85,B 0,C 180,E1 -14829.467,E2 -14829.467} C_VEL
LIN {X 0,Y 328.077,Z 570.187,A -85,B 0,C 180,E1 -14831.907,E2 -14831.907} C_VEL
LIN {X 0,Y 326.858,Z 578.462,A -85,B 0,C 180,E1 -14834.412,E2 -14834.412} C_VEL
LIN {X 0,Y 326.162,Z 585.296,A -85,B 0,C 180,E1 -14836.927,E2 -14836.927} C_VEL
LIN {X 0,Y 325.725,Z 590.768,A -85,B 0,C 180,E1 -14839.435,E2 -14839.435} C_VEL
LIN {X 0,Y 325.596,Z 594.045,A -85,B 0,C 180,E1 -14841.313,E2 -14841.313} C_VEL
LIN {X 0,Y 325.578,Z 597.361,A -85,B 0,C 180,E1 -14843.807,E2 -14843.807} C_VEL
LIN {X 0,Y 325.749,Z 599.547,A -85,B 0,C 180,E1 -14846.292,E2 -14846.292} C_VEL
LIN {X 0,Y 325.676,Z 600.607,A -85,B 0,C 180,E1 -14848.767,E2 -14848.767} C_VEL
LIN {X 0,Y 325.687,Z 600.506,A -85,B 0,C 180,E1 -14851.239,E2 -14851.239} C_VEL
LIN {X 0,Y 325.763,Z 599.386,A -85,B 0,C 180,E1 -14853.714,E2 -14853.714} C_VEL
LIN {X 0,Y 325.607,Z 597.058,A -85,B 0,C 180,E1 -14856.198,E2 -14856.198} C_VEL
LIN {X 0,Y 325.646,Z 593.668,A -85,B 0,C 180,E1 -14858.692,E2 -14858.692} C_VEL
LIN {X 0,Y 325.786,Z 589.121,A -85,B 0,C 180,E1 -14861.198,E2 -14861.198} C_VEL
LIN {X 0,Y 326.326,Z 583.365,A -85,B 0,C 180,E1 -14863.707,E2 -14863.707} C_VEL
LIN {X 0,Y 327.106,Z 576.384,A -85,B 0,C 180,E1 -14866.222,E2 -14866.222} C_VEL
LIN {X 0,Y 328.338,Z 568.032,A -85,B 0,C 180,E1 -14868.73,E2 -14868.73} C_VEL
LIN {X 0,Y 330.08,Z 558.128,A -85,B 0,C 180,E1 -14871.223,E2 -14871.223} C_VEL
LIN {X 0,Y 332.054,Z 548.058,A -85,B 0,C 180,E1 -14873.384,E2 -14873.384} C_VEL
LIN {X 0,Y 334.525,Z 536.343,A -85,B 0,C 180,E1 -14875.541,E2 -14875.541} C_VEL
LIN {X 0,Y 337.343,Z 523.09,A -85,B 0,C 180,E1 -14877.619,E2 -14877.619} C_VEL
LIN {X 0,Y 340.504,Z 508.597,A -85,B 0,C 180,E1 -14879.526,E2 -14879.526} C_VEL
LIN {X 0,Y 343.508,Z 494.341,A -85,B 0,C 180,E1 -14881.107,E2 -14881.107} C_VEL
LIN {X 0,Y 346.655,Z 479.14,A -85,B 0,C 180,E1 -14882.499,E2 -14882.499} C_VEL
LIN {X 0,Y 348.498,Z 469.144,A -85,B 0,C 180,E1 -14883.288,E2 -14883.288} C_VEL
LIN {X 0,Y 348.528,Z 455.434,A -85,B 0,C 180,E1 -14884.545,E2 -14884.545} C_VEL
LIN {X 0,Y 348.521,Z 442.02,A -85,B 0,C 180,E1 -14885.648,E2 -14885.648} C_VEL
LIN {X 0,Y 347.433,Z 429.649,A -85,B 0,C 180,E1 -14886.75,E2 -14886.75} C_VEL
LIN {X 0,Y 345.025,Z 415.797,A -85,B 0,C 180,E1 -14888.177,E2 -14888.177} C_VEL
LIN {X 0,Y 343.914,Z 410.74,A -85,B 0,C 180,E1 -14888.784,E2 -14888.784} C_VEL
LIN {X 0,Y 343.386,Z 407.511,A -85,B 0,C 180,E1 -14889.155,E2 -14889.155} C_VEL
LIN {X 0,Y 345.229,Z 403.166,A -85,B 0,C 180,E1 -14890.653,E2 -14890.653} C_VEL
LIN {X 0,Y 344.392,Z 399.372,A -85,B 0,C 180,E1 -14892.723,E2 -14892.723} C_VEL
LIN {X 0,Y 343.581,Z 397.059,A -85,B 0,C 180,E1 -14894.281,E2 -14894.281} C_VEL
LIN {X 0,Y 342.878,Z 395.164,A -85,B 0,C 180,E1 -14895.843,E2 -14895.843} C_VEL
LIN {X 0,Y 341.597,Z 392.627,A -85,B 0,C 180,E1 -14898.825,E2 -14898.825} C_VEL
LIN {X 0,Y 341.005,Z 391.882,A -85,B 0,C 180,E1 -14900.291,E2 -14900.291} C_VEL
LIN {X 0,Y 340.321,Z 391.49,A -85,B 0,C 180,E1 -14901.718,E2 -14901.718} C_VEL
LIN {X 0,Y 338.721,Z 391.658,A -85,B 0,C 180,E1 -14904.482,E2 -14904.482} C_VEL
LIN {X 0,Y 336.561,Z 393.163,A -85,B 0,C 180,E1 -14907.981,E2 -14907.981} C_VEL
LIN {X 0,Y 337.386,Z 395.469,A -85,B 0,C 180,E1 -14908.659,E2 -14908.659} C_VEL
LIN {X 0,Y 338.96,Z 397.958,A -85,B 0,C 180,E1 -14909.561,E2 -14909.561} C_VEL
LIN {X 0,Y 342.196,Z 404.669,A -85,B 0,C 180,E1 -14911.424,E2 -14911.424} C_VEL
LIN {X 0,Y 345.775,Z 413.424,A -85,B 0,C 180,E1 -14913.439,E2 -14913.439} C_VEL
LIN {X 0,Y 348.679,Z 423.446,A -85,B 0,C 180,E1 -14915.388,E2 -14915.388} C_VEL
LIN {X 0,Y 349.425,Z 426.903,A -85,B 0,C 180,E1 -14916.002,E2 -14916.002} C_VEL
LIN {X 0,Y 346.28,Z 441.426,A -85,B 0,C 180,E1 -14917.633,E2 -14917.633} C_VEL
LIN {X 0,Y 343.796,Z 451.89,A -85,B 0,C 180,E1 -14919.039,E2 -14919.039} C_VEL
LIN {X 0,Y 341.151,Z 462.585,A -85,B 0,C 180,E1 -14920.755,E2 -14920.755} C_VEL
LIN {X 0,Y 338.783,Z 471.571,A -85,B 0,C 180,E1 -14922.495,E2 -14922.495} C_VEL
LIN {X 0,Y 336.479,Z 480.004,A -85,B 0,C 180,E1 -14924.482,E2 -14924.482} C_VEL
LIN {X 0,Y 334.327,Z 487.332,A -85,B 0,C 180,E1 -14926.631,E2 -14926.631} C_VEL
LIN {X 0,Y 332.693,Z 492.204,A -85,B 0,C 180,E1 -14928.424,E2 -14928.424} C_VEL
LIN {X 0,Y 331.332,Z 496.045,A -85,B 0,C 180,E1 -14930.231,E2 -14930.231} C_VEL
LIN {X 0,Y 330.596,Z 498.067,A -85,B 0,C 180,E1 -14931.443,E2 -14931.443} C_VEL
LIN {X 0,Y 330.009,Z 499.659,A -85,B 0,C 180,E1 -14932.659,E2 -14932.659} C_VEL
LIN {X 0,Y 329.559,Z 500.822,A -85,B 0,C 180,E1 -14933.88,E2 -14933.88} C_VEL
LIN {X 0,Y 329.039,Z 501.612,A -85,B 0,C 180,E1 -14935.099,E2 -14935.099} C_VEL
LIN {X 0,Y 328.608,Z 502.001,A -85,B 0,C 180,E1 -14936.322,E2 -14936.322} C_VEL
LIN {X 0,Y 328.162,Z 502.012,A -85,B 0,C 180,E1 -14937.546,E2 -14937.546} C_VEL
LIN {X 0,Y 327.886,Z 501.605,A -85,B 0,C 180,E1 -14938.772,E2 -14938.772} C_VEL
LIN {X 0,Y 327.657,Z 500.8,A -85,B 0,C 180,E1 -14940,E2 -14940} C_VEL
LIN {X 0,Y 327.528,Z 499.554,A -85,B 0,C 180,E1 -14941.23,E2 -14941.23} C_VEL
LIN {X 0,Y 327.452,Z 496.92,A -85,B 0,C 180,E1 -14943.076,E2 -14943.076} C_VEL
LIN {X 0,Y 327.456,Z 493.303,A -85,B 0,C 180,E1 -14944.925,E2 -14944.925} C_VEL
LIN {X 0,Y 327.63,Z 488.657,A -85,B 0,C 180,E1 -14946.776,E2 -14946.776} C_VEL
LIN {X 0,Y 328.179,Z 482.866,A -85,B 0,C 180,E1 -14948.622,E2 -14948.622} C_VEL
LIN {X 0,Y 328.714,Z 474.548,A -85,B 0,C 180,E1 -14950.782,E2 -14950.782} C_VEL
LIN {X 0,Y 329.445,Z 465.812,A -85,B 0,C 180,E1 -14952.631,E2 -14952.631} C_VEL
LIN {X 0,Y 330.265,Z 455.324,A -85,B 0,C 180,E1 -14954.48,E2 -14954.48} C_VEL
LIN {X 0,Y 331.458,Z 443.686,A -85,B 0,C 180,E1 -14956.159,E2 -14956.159} C_VEL
LIN {X 0,Y 332.487,Z 430.933,A -85,B 0,C 180,E1 -14957.691,E2 -14957.691} C_VEL
LIN {X 0,Y 333.409,Z 418.589,A -85,B 0,C 180,E1 -14958.911,E2 -14958.911} C_VEL
LIN {X 0,Y 334.483,Z 405.711,A -85,B 0,C 180,E1 -14959.936,E2 -14959.936} C_VEL
LIN {X 0,Y 331.863,Z 392.886,A -85,B 0,C 180,E1 -14960.963,E2 -14960.963} C_VEL
LIN {X 0,Y 328.185,Z 377.668,A -85,B 0,C 180,E1 -14961.984,E2 -14961.984} C_VEL
LIN {X 0,Y 326.927,Z 372.484,A -85,B 0,C 180,E1 -14962.291,E2 -14962.291} C_VEL
LIN {X 0,Y 327.222,Z 366.1,A -85,B 0,C 180,E1 -14966.123,E2 -14966.123} C_VEL
LIN {X 0,Y 327.573,Z 360.466,A -85,B 0,C 180,E1 -14969.569,E2 -14969.569} C_VEL
LIN {X 0,Y 327.933,Z 354.554,A -85,B 0,C 180,E1 -14973.296,E2 -14973.296} C_VEL
LIN {X 0,Y 328.116,Z 350.199,A -85,B 0,C 180,E1 -14976.111,E2 -14976.111} C_VEL
LIN {X 0,Y 327.759,Z 346.763,A -85,B 0,C 180,E1 -14978.451,E2 -14978.451} C_VEL
LIN {X 0,Y 326.983,Z 342.028,A -85,B 0,C 180,E1 -14981.783,E2 -14981.783} C_VEL
LIN {X 0,Y 326.609,Z 340.113,A -85,B 0,C 180,E1 -14983.28,E2 -14983.28} C_VEL
LIN {X 0,Y 326.588,Z 340.327,A -85,B 0,C 180,E1 -14984.641,E2 -14984.641} C_VEL
LIN {X 0,Y 328.391,Z 348.071,A -85,B 0,C 180,E1 -14988.434,E2 -14988.434} C_VEL
LIN {X 0,Y 329.734,Z 355.315,A -85,B 0,C 180,E1 -14992.058,E2 -14992.058} C_VEL
LIN {X 0,Y 330.231,Z 359.343,A -85,B 0,C 180,E1 -14993.972,E2 -14993.972} C_VEL
LIN {X 0,Y 330.06,Z 367.534,A -85,B 0,C 180,E1 -14997.835,E2 -14997.835} C_VEL
LIN {X 0,Y 329.91,Z 376.683,A -85,B 0,C 180,E1 -15002.05,E2 -15002.05} C_VEL
LIN {X 0,Y 330.061,Z 386.089,A -85,B 0,C 180,E1 -15006.133,E2 -15006.133} C_VEL
LIN {X 0,Y 330.209,Z 390.961,A -85,B 0,C 180,E1 -15008.011,E2 -15008.011} C_VEL
LIN {X 0,Y 334.614,Z 403.691,A -85,B 0,C 180,E1 -15008.77,E2 -15008.77} C_VEL
LIN {X 0,Y 336.595,Z 411.155,A -85,B 0,C 180,E1 -15009.3,E2 -15009.3} C_VEL
LIN {X 0,Y 336.046,Z 423.349,A -85,B 0,C 180,E1 -15010.088,E2 -15010.088} C_VEL
LIN {X 0,Y 335.287,Z 433.983,A -85,B 0,C 180,E1 -15010.995,E2 -15010.995} C_VEL
LIN {X 0,Y 334.37,Z 444.179,A -85,B 0,C 180,E1 -15012.095,E2 -15012.095} C_VEL
LIN {X 0,Y 333.057,Z 455.378,A -85,B 0,C 180,E1 -15013.604,E2 -15013.604} C_VEL
LIN {X 0,Y 332.132,Z 463.512,A -85,B 0,C 180,E1 -15014.974,E2 -15014.974} C_VEL
LIN {X 0,Y 331.071,Z 471.027,A -85,B 0,C 180,E1 -15016.494,E2 -15016.494} C_VEL
LIN {X 0,Y 330.215,Z 477.338,A -85,B 0,C 180,E1 -15018.05,E2 -15018.05} C_VEL
LIN {X 0,Y 329.544,Z 482.363,A -85,B 0,C 180,E1 -15019.553,E2 -15019.553} C_VEL
LIN {X 0,Y 328.598,Z 487.413,A -85,B 0,C 180,E1 -15021.387,E2 -15021.387} C_VEL
LIN {X 0,Y 327.939,Z 491.305,A -85,B 0,C 180,E1 -15023.228,E2 -15023.228} C_VEL
LIN {X 0,Y 327.648,Z 494.141,A -85,B 0,C 180,E1 -15025.075,E2 -15025.075} C_VEL
LIN {X 0,Y 327.426,Z 495.529,A -85,B 0,C 180,E1 -15026.305,E2 -15026.305} C_VEL
LIN {X 0,Y 327.062,Z 497.119,A -85,B 0,C 180,E1 -15028.766,E2 -15028.766} C_VEL
LIN {X 0,Y 327.047,Z 497.346,A -85,B 0,C 180,E1 -15029.997,E2 -15029.997} C_VEL
LIN {X 0,Y 327.182,Z 496.583,A -85,B 0,C 180,E1 -15032.459,E2 -15032.459} C_VEL
LIN {X 0,Y 327.437,Z 495.622,A -85,B 0,C 180,E1 -15033.689,E2 -15033.689} C_VEL
LIN {X 0,Y 327.671,Z 494.286,A -85,B 0,C 180,E1 -15034.919,E2 -15034.919} C_VEL
LIN {X 0,Y 327.92,Z 491.511,A -85,B 0,C 180,E1 -15036.766,E2 -15036.766} C_VEL
LIN {X 0,Y 328.585,Z 487.685,A -85,B 0,C 180,E1 -15038.608,E2 -15038.608} C_VEL
LIN {X 0,Y 329.498,Z 482.711,A -85,B 0,C 180,E1 -15040.442,E2 -15040.442} C_VEL
LIN {X 0,Y 330.317,Z 476.476,A -85,B 0,C 180,E1 -15042.281,E2 -15042.281} C_VEL
LIN {X 0,Y 331.402,Z 468.696,A -85,B 0,C 180,E1 -15044.112,E2 -15044.112} C_VEL
LIN {X 0,Y 332.526,Z 460.715,A -85,B 0,C 180,E1 -15045.63,E2 -15045.63} C_VEL
LIN {X 0,Y 333.528,Z 452.011,A -85,B 0,C 180,E1 -15046.996,E2 -15046.996} C_VEL
LIN {X 0,Y 334.584,Z 441.206,A -85,B 0,C 180,E1 -15048.362,E2 -15048.362} C_VEL
LIN {X 0,Y 335.611,Z 429.963,A -85,B 0,C 180,E1 -15049.477,E2 -15049.477} C_VEL
LIN {X 0,Y 336.317,Z 418.858,A -85,B 0,C 180,E1 -15050.338,E2 -15050.338} C_VEL
LIN {X 0,Y 336.55,Z 410.455,A -85,B 0,C 180,E1 -15050.851,E2 -15050.851} C_VEL
LIN {X 0,Y 332.815,Z 398.041,A -85,B 0,C 180,E1 -15051.697,E2 -15051.697} C_VEL
LIN {X 0,Y 330.185,Z 390.726,A -85,B 0,C 180,E1 -15052.12,E2 -15052.12} C_VEL
LIN {X 0,Y 329.986,Z 381.643,A -85,B 0,C 180,E1 -15055.876,E2 -15055.876} C_VEL
LIN {X 0,Y 329.981,Z 372.366,A -85,B 0,C 180,E1 -15060.029,E2 -15060.029} C_VEL
LIN {X 0,Y 330.155,Z 364.186,A -85,B 0,C 180,E1 -15063.881,E2 -15063.881} C_VEL
LIN {X 0,Y 330.239,Z 359.644,A -85,B 0,C 180,E1 -15066.03,E2 -15066.03} C_VEL
LIN {X 0,Y 329.717,Z 355.238,A -85,B 0,C 180,E1 -15068.176,E2 -15068.176} C_VEL
LIN {X 0,Y 328.858,Z 350.319,A -85,B 0,C 180,E1 -15070.671,E2 -15070.671} C_VEL
LIN {X 0,Y 327.32,Z 343.185,A -85,B 0,C 180,E1 -15074.082,E2 -15074.082} C_VEL
LIN {X 0,Y 326.623,Z 340.113,A -85,B 0,C 180,E1 -15075.612,E2 -15075.612} C_VEL
LIN {X 0,Y 326.608,Z 340.116,A -85,B 0,C 180,E1 -15076.888,E2 -15076.888} C_VEL
LIN {X 0,Y 325.983,Z 340.198,A -85,B 0,C 180,E1 -15077.917,E2 -15077.917} C_VEL
LIN {X 0,Y 323.188,Z 340.549,A -85,B 0,C 180,E1 -15079.594,E2 -15079.594} C_VEL
LIN {X 0,Y 320.771,Z 340.846,A -85,B 0,C 180,E1 -15080.952,E2 -15080.952} C_VEL
LIN {X 0,Y 319.691,Z 340.976,A -85,B 0,C 180,E1 -15082.002,E2 -15082.002} C_VEL
LIN {X 0,Y 319.581,Z 340.987,A -85,B 0,C 180,E1 -15082.358,E2 -15082.358} C_VEL
LIN {X 0,Y 319.543,Z 340.994,A -85,B 0,C 180,E1 -15085.121,E2 -15085.121} C_VEL
LIN {X 0,Y 319.552,Z 340.992,A -85,B 0,C 180,E1 -15089.055,E2 -15089.055} C_VEL
LIN {X 0,Y 319.589,Z 340.985,A -85,B 0,C 180,E1 -15092.496,E2 -15092.496} C_VEL
LIN {X 0,Y 319.607,Z 340.986,A -85,B 0,C 180,E1 -15095.304,E2 -15095.304} C_VEL
LIN {X 0,Y 319.605,Z 340.98,A -85,B 0,C 180,E1 -15098.048,E2 -15098.048} C_VEL
LIN {X 0,Y 319.685,Z 340.967,A -85,B 0,C 180,E1 -15100.951,E2 -15100.951} C_VEL
LIN {X 0,Y 319.709,Z 340.961,A -85,B 0,C 180,E1 -15105.274,E2 -15105.274} C_VEL
LIN {X 0,Y 319.738,Z 340.959,A -85,B 0,C 180,E1 -15109.872,E2 -15109.872} C_VEL
LIN {X 0,Y 319.91,Z 340.949,A -85,B 0,C 180,E1 -15112.425,E2 -15112.425} C_VEL
LIN {X 0,Y 319.722,Z 340.961,A -85,B 0,C 180,E1 -15114.955,E2 -15114.955} C_VEL
LIN {X 0,Y 319.965,Z 340.942,A -85,B 0,C 180,E1 -15117.482,E2 -15117.482} C_VEL
LIN {X 0,Y 320.108,Z 340.913,A -85,B 0,C 180,E1 -15120,E2 -15120} C_VEL
LIN {X 0,Y 319.997,Z 340.935,A -85,B 0,C 180,E1 -15122.517,E2 -15122.517} C_VEL
LIN {X 0,Y 319.932,Z 340.944,A -85,B 0,C 180,E1 -15126.305,E2 -15126.305} C_VEL
LIN {X 0,Y 319.819,Z 340.96,A -85,B 0,C 180,E1 -15128.848,E2 -15128.848} C_VEL
LIN {X 0,Y 319.662,Z 340.98,A -85,B 0,C 180,E1 -15132.7,E2 -15132.7} C_VEL
LIN {X 0,Y 319.677,Z 340.978,A -85,B 0,C 180,E1 -15135.296,E2 -15135.296} C_VEL
LIN {X 0,Y 319.669,Z 340.979,A -85,B 0,C 180,E1 -15139.255,E2 -15139.255} C_VEL
LIN {X 0,Y 319.623,Z 340.982,A -85,B 0,C 180,E1 -15143.315,E2 -15143.315} C_VEL
LIN {X 0,Y 319.614,Z 340.983,A -85,B 0,C 180,E1 -15146.089,E2 -15146.089} C_VEL
LIN {X 0,Y 319.611,Z 341.059,A -85,B 0,C 180,E1 -15148.135,E2 -15148.135} C_VEL
LIN {X 0,Y 321.534,Z 348.354,A -85,B 0,C 180,E1 -15151.64,E2 -15151.64} C_VEL
LIN {X 0,Y 323.82,Z 356.077,A -85,B 0,C 180,E1 -15155.109,E2 -15155.109} C_VEL
LIN {X 0,Y 326.624,Z 366.144,A -85,B 0,C 180,E1 -15159.236,E2 -15159.236} C_VEL
LIN {X 0,Y 329.462,Z 376.28,A -85,B 0,C 180,E1 -15163.048,E2 -15163.048} C_VEL
LIN {X 0,Y 332.258,Z 385.901,A -85,B 0,C 180,E1 -15166.41,E2 -15166.41} C_VEL
LIN {X 0,Y 335,Z 396.517,A -85,B 0,C 180,E1 -15169.831,E2 -15169.831} C_VEL
LIN {X 0,Y 331.503,Z 410.913,A -85,B 0,C 180,E1 -15173.591,E2 -15173.591} C_VEL
LIN {X 0,Y 330.917,Z 413.624,A -85,B 0,C 180,E1 -15174.293,E2 -15174.293} C_VEL
LIN {X 0,Y 334.316,Z 436.169,A -85,B 0,C 180,E1 -15175.356,E2 -15175.356} C_VEL
LIN {X 0,Y 336.522,Z 452.147,A -85,B 0,C 180,E1 -15176.302,E2 -15176.302} C_VEL
LIN {X 0,Y 338.179,Z 467.445,A -85,B 0,C 180,E1 -15177.387,E2 -15177.387} C_VEL
LIN {X 0,Y 336.161,Z 483.05,A -85,B 0,C 180,E1 -15178.493,E2 -15178.493} C_VEL
LIN {X 0,Y 333.738,Z 498.215,A -85,B 0,C 180,E1 -15179.821,E2 -15179.821} C_VEL
LIN {X 0,Y 331.468,Z 512.327,A -85,B 0,C 180,E1 -15181.338,E2 -15181.338} C_VEL
LIN {X 0,Y 329,Z 525.399,A -85,B 0,C 180,E1 -15183.008,E2 -15183.008} C_VEL
LIN {X 0,Y 326.684,Z 537.614,A -85,B 0,C 180,E1 -15184.861,E2 -15184.861} C_VEL
LIN {X 0,Y 324.436,Z 549.717,A -85,B 0,C 180,E1 -15187.054,E2 -15187.054} C_VEL
LIN {X 0,Y 322.556,Z 559.936,A -85,B 0,C 180,E1 -15189.268,E2 -15189.268} C_VEL
LIN {X 0,Y 321.002,Z 569.825,A -85,B 0,C 180,E1 -15191.824,E2 -15191.824} C_VEL
LIN {X 0,Y 319.907,Z 577.066,A -85,B 0,C 180,E1 -15194.065,E2 -15194.065} C_VEL
LIN {X 0,Y 319.159,Z 583.993,A -85,B 0,C 180,E1 -15196.635,E2 -15196.635} C_VEL
LIN {X 0,Y 318.704,Z 589.508,A -85,B 0,C 180,E1 -15199.2,E2 -15199.2} C_VEL
LIN {X 0,Y 318.569,Z 592.858,A -85,B 0,C 180,E1 -15201.12,E2 -15201.12} C_VEL
LIN {X 0,Y 318.553,Z 596.205,A -85,B 0,C 180,E1 -15203.67,E2 -15203.67} C_VEL
LIN {X 0,Y 318.721,Z 598.439,A -85,B 0,C 180,E1 -15206.21,E2 -15206.21} C_VEL
LIN {X 0,Y 318.658,Z 599.516,A -85,B 0,C 180,E1 -15208.739,E2 -15208.739} C_VEL
LIN {X 0,Y 318.662,Z 599.451,A -85,B 0,C 180,E1 -15211.267,E2 -15211.267} C_VEL
LIN {X 0,Y 318.736,Z 598.356,A -85,B 0,C 180,E1 -15213.796,E2 -15213.796} C_VEL
LIN {X 0,Y 318.625,Z 595.318,A -85,B 0,C 180,E1 -15216.99,E2 -15216.99} C_VEL
LIN {X 0,Y 318.58,Z 591.614,A -85,B 0,C 180,E1 -15219.526,E2 -15219.526} C_VEL
LIN {X 0,Y 318.881,Z 586.823,A -85,B 0,C 180,E1 -15222.089,E2 -15222.089} C_VEL
LIN {X 0,Y 319.525,Z 580.445,A -85,B 0,C 180,E1 -15224.803,E2 -15224.803} C_VEL
LIN {X 0,Y 320.489,Z 573.505,A -85,B 0,C 180,E1 -15227.223,E2 -15227.223} C_VEL
LIN {X 0,Y 321.855,Z 565.073,A -85,B 0,C 180,E1 -15229.725,E2 -15229.725} C_VEL
LIN {X 0,Y 323.866,Z 554.687,A -85,B 0,C 180,E1 -15232.321,E2 -15232.321} C_VEL
LIN {X 0,Y 326.448,Z 542.764,A -85,B 0,C 180,E1 -15234.825,E2 -15234.825} C_VEL
LIN {X 0,Y 329.207,Z 530.647,A -85,B 0,C 180,E1 -15236.981,E2 -15236.981} C_VEL
LIN {X 0,Y 332.482,Z 516.599,A -85,B 0,C 180,E1 -15239.092,E2 -15239.092} C_VEL
LIN {X 0,Y 335.84,Z 502.16,A -85,B 0,C 180,E1 -15240.909,E2 -15240.909} C_VEL
LIN {X 0,Y 339.031,Z 487.696,A -85,B 0,C 180,E1 -15242.44,E2 -15242.44} C_VEL
LIN {X 0,Y 342.703,Z 470.309,A -85,B 0,C 180,E1 -15243.952,E2 -15243.952} C_VEL
LIN {X 0,Y 343.021,Z 457.144,A -85,B 0,C 180,E1 -15245.224,E2 -15245.224} C_VEL
LIN {X 0,Y 343.33,Z 443.621,A -85,B 0,C 180,E1 -15246.418,E2 -15246.418} C_VEL
LIN {X 0,Y 342.359,Z 430.45,A -85,B 0,C 180,E1 -15247.688,E2 -15247.688} C_VEL
LIN {X 0,Y 340.558,Z 418.354,A -85,B 0,C 180,E1 -15249.04,E2 -15249.04} C_VEL
LIN {X 0,Y 339.072,Z 410.587,A -85,B 0,C 180,E1 -15250.048,E2 -15250.048} C_VEL
LIN {X 0,Y 338.451,Z 406.357,A -85,B 0,C 180,E1 -15250.659,E2 -15250.659} C_VEL
LIN {X 0,Y 338.651,Z 405.909,A -85,B 0,C 180,E1 -15250.826,E2 -15250.826} C_VEL
LIN {X 0,Y 338.132,Z 402.879,A -85,B 0,C 180,E1 -15252.461,E2 -15252.461} C_VEL
LIN {X 0,Y 336.755,Z 399.054,A -85,B 0,C 180,E1 -15255.203,E2 -15255.203} C_VEL
LIN {X 0,Y 335.581,Z 396.387,A -85,B 0,C 180,E1 -15257.921,E2 -15257.921} C_VEL
LIN {X 0,Y 334.99,Z 395.372,A -85,B 0,C 180,E1 -15259.431,E2 -15259.431} C_VEL
LIN {X 0,Y 334.169,Z 394.714,A -85,B 0,C 180,E1 -15261.095,E2 -15261.095} C_VEL
LIN {X 0,Y 332.732,Z 394.521,A -85,B 0,C 180,E1 -15263.743,E2 -15263.743} C_VEL
LIN {X 0,Y 331.347,Z 395.143,A -85,B 0,C 180,E1 -15265.816,E2 -15265.816} C_VEL
LIN {X 0,Y 332.038,Z 397.249,A -85,B 0,C 180,E1 -15266.611,E2 -15266.611} C_VEL
LIN {X 0,Y 333.236,Z 399.07,A -85,B 0,C 180,E1 -15267.526,E2 -15267.526} C_VEL
LIN {X 0,Y 335.496,Z 403.8,A -85,B 0,C 180,E1 -15269.194,E2 -15269.194} C_VEL
LIN {X 0,Y 337.977,Z 409.436,A -85,B 0,C 180,E1 -15270.855,E2 -15270.855} C_VEL
LIN {X 0,Y 340.724,Z 416.861,A -85,B 0,C 180,E1 -15272.71,E2 -15272.71} C_VEL
LIN {X 0,Y 342.601,Z 423.39,A -85,B 0,C 180,E1 -15274.106,E2 -15274.106} C_VEL
LIN {X 0,Y 344.038,Z 429.963,A -85,B 0,C 180,E1 -15275.386,E2 -15275.386} C_VEL
LIN {X 0,Y 340.309,Z 445.494,A -85,B 0,C 180,E1 -15277.219,E2 -15277.219} C_VEL
LIN {X 0,Y 337.231,Z 457.234,A -85,B 0,C 180,E1 -15278.931,E2 -15278.931} C_VEL
LIN {X 0,Y 334.516,Z 467.114,A -85,B 0,C 180,E1 -15280.677,E2 -15280.677} C_VEL
LIN {X 0,Y 332.059,Z 475.698,A -85,B 0,C 180,E1 -15282.479,E2 -15282.479} C_VEL
LIN {X 0,Y 329.581,Z 483.759,A -85,B 0,C 180,E1 -15284.541,E2 -15284.541} C_VEL
LIN {X 0,Y 327.749,Z 489.477,A -85,B 0,C 180,E1 -15286.357,E2 -15286.357} C_VEL
LIN {X 0,Y 325.496,Z 495.504,A -85,B 0,C 180,E1 -15288.795,E2 -15288.795} C_VEL
LIN {X 0,Y 324.584,Z 497.846,A -85,B 0,C 180,E1 -15290.025,E2 -15290.025} C_VEL
LIN {X 0,Y 323.167,Z 501.281,A -85,B 0,C 180,E1 -15292.503,E2 -15292.503} C_VEL
LIN {X 0,Y 322.67,Z 502.349,A -85,B 0,C 180,E1 -15293.748,E2 -15293.748} C_VEL
LIN {X 0,Y 321.667,Z 503.361,A -85,B 0,C 180,E1 -15296.242,E2 -15296.242} C_VEL
LIN {X 0,Y 321.205,Z 503.309,A -85,B 0,C 180,E1 -15297.492,E2 -15297.492} C_VEL
LIN {X 0,Y 320.911,Z 502.838,A -85,B 0,C 180,E1 -15298.746,E2 -15298.746} C_VEL
LIN {X 0,Y 320.653,Z 501.946,A -85,B 0,C 180,E1 -15300,E2 -15300} C_VEL
LIN {X 0,Y 320.523,Z 500.617,A -85,B 0,C 180,E1 -15301.257,E2 -15301.257} C_VEL
LIN {X 0,Y 320.455,Z 497.883,A -85,B 0,C 180,E1 -15303.143,E2 -15303.143} C_VEL
LIN {X 0,Y 320.449,Z 494.165,A -85,B 0,C 180,E1 -15305.033,E2 -15305.033} C_VEL
LIN {X 0,Y 320.615,Z 489.398,A -85,B 0,C 180,E1 -15306.925,E2 -15306.925} C_VEL
LIN {X 0,Y 321.238,Z 482.439,A -85,B 0,C 180,E1 -15309.111,E2 -15309.111} C_VEL
LIN {X 0,Y 321.87,Z 473.659,A -85,B 0,C 180,E1 -15311.334,E2 -15311.334} C_VEL
LIN {X 0,Y 322.668,Z 464.529,A -85,B 0,C 180,E1 -15313.221,E2 -15313.221} C_VEL
LIN {X 0,Y 323.577,Z 453.477,A -85,B 0,C 180,E1 -15315.108,E2 -15315.108} C_VEL
LIN {X 0,Y 324.78,Z 441.29,A -85,B 0,C 180,E1 -15316.824,E2 -15316.824} C_VEL
LIN {X 0,Y 325.866,Z 427.802,A -85,B 0,C 180,E1 -15318.38,E2 -15318.38} C_VEL
LIN {X 0,Y 327.021,Z 414.572,A -85,B 0,C 180,E1 -15319.621,E2 -15319.621} C_VEL
LIN {X 0,Y 327.668,Z 406.673,A -85,B 0,C 180,E1 -15320.241,E2 -15320.241} C_VEL
LIN {X 0,Y 324.635,Z 392.306,A -85,B 0,C 180,E1 -15321.419,E2 -15321.419} C_VEL
LIN {X 0,Y 320.894,Z 376.838,A -85,B 0,C 180,E1 -15322.465,E2 -15322.465} C_VEL
LIN {X 0,Y 319.924,Z 372.868,A -85,B 0,C 180,E1 -15322.731,E2 -15322.731} C_VEL
LIN {X 0,Y 320.258,Z 366.268,A -85,B 0,C 180,E1 -15326.736,E2 -15326.736} C_VEL
LIN {X 0,Y 320.606,Z 360.596,A -85,B 0,C 180,E1 -15330.278,E2 -15330.278} C_VEL
LIN {X 0,Y 320.99,Z 355.236,A -85,B 0,C 180,E1 -15333.691,E2 -15333.691} C_VEL
LIN {X 0,Y 321.15,Z 351.389,A -85,B 0,C 180,E1 -15336.219,E2 -15336.219} C_VEL
LIN {X 0,Y 320.553,Z 346.692,A -85,B 0,C 180,E1 -15339.481,E2 -15339.481} C_VEL
LIN {X 0,Y 319.748,Z 341.869,A -85,B 0,C 180,E1 -15342.952,E2 -15342.952} C_VEL
LIN {X 0,Y 319.556,Z 340.994,A -85,B 0,C 180,E1 -15343.786,E2 -15343.786} C_VEL
LIN {X 0,Y 321.184,Z 348.101,A -85,B 0,C 180,E1 -15347.284,E2 -15347.284} C_VEL
LIN {X 0,Y 322.381,Z 354.087,A -85,B 0,C 180,E1 -15350.296,E2 -15350.296} C_VEL
LIN {X 0,Y 323.306,Z 359.773,A -85,B 0,C 180,E1 -15353.112,E2 -15353.112} C_VEL
LIN {X 0,Y 323.359,Z 365.172,A -85,B 0,C 180,E1 -15355.681,E2 -15355.681} C_VEL
LIN {X 0,Y 323.13,Z 372.771,A -85,B 0,C 180,E1 -15359.259,E2 -15359.259} C_VEL
LIN {X 0,Y 323.144,Z 381.2,A -85,B 0,C 180,E1 -15363.089,E2 -15363.089} C_VEL
LIN {X 0,Y 323.298,Z 388.469,A -85,B 0,C 180,E1 -15366.194,E2 -15366.194} C_VEL
LIN {X 0,Y 323.351,Z 391.719,A -85,B 0,C 180,E1 -15367.503,E2 -15367.503} C_VEL
LIN {X 0,Y 327.938,Z 405.014,A -85,B 0,C 180,E1 -15368.329,E2 -15368.329} C_VEL
LIN {X 0,Y 330.016,Z 412.695,A -85,B 0,C 180,E1 -15368.896,E2 -15368.896} C_VEL
LIN {X 0,Y 329.447,Z 424.594,A -85,B 0,C 180,E1 -15369.687,E2 -15369.687} C_VEL
LIN {X 0,Y 328.575,Z 436.08,A -85,B 0,C 180,E1 -15370.703,E2 -15370.703} C_VEL
LIN {X 0,Y 327.698,Z 445.248,A -85,B 0,C 180,E1 -15371.718,E2 -15371.718} C_VEL
LIN {X 0,Y 326.329,Z 456.45,A -85,B 0,C 180,E1 -15373.256,E2 -15373.256} C_VEL
LIN {X 0,Y 325.364,Z 464.585,A -85,B 0,C 180,E1 -15374.654,E2 -15374.654} C_VEL
LIN {X 0,Y 324.271,Z 472.099,A -85,B 0,C 180,E1 -15376.205,E2 -15376.205} C_VEL
LIN {X 0,Y 323.352,Z 478.389,A -85,B 0,C 180,E1 -15377.785,E2 -15377.785} C_VEL
LIN {X 0,Y 322.65,Z 483.439,A -85,B 0,C 180,E1 -15379.327,E2 -15379.327} C_VEL
LIN {X 0,Y 321.66,Z 488.49,A -85,B 0,C 180,E1 -15381.2,E2 -15381.2} C_VEL
LIN {X 0,Y 320.968,Z 492.382,A -85,B 0,C 180,E1 -15383.08,E2 -15383.08} C_VEL
LIN {X 0,Y 320.664,Z 495.218,A -85,B 0,C 180,E1 -15384.968,E2 -15384.968} C_VEL
LIN {X 0,Y 320.424,Z 496.606,A -85,B 0,C 180,E1 -15386.224,E2 -15386.224} C_VEL
LIN {X 0,Y 320.065,Z 498.193,A -85,B 0,C 180,E1 -15388.739,E2 -15388.739} C_VEL
LIN {X 0,Y 320.044,Z 498.42,A -85,B 0,C 180,E1 -15389.997,E2 -15389.997} C_VEL
LIN {X 0,Y 320.171,Z 497.659,A -85,B 0,C 180,E1 -15392.513,E2 -15392.513} C_VEL
LIN {X 0,Y 320.434,Z 496.698,A -85,B 0,C 180,E1 -15393.77,E2 -15393.77} C_VEL
LIN {X 0,Y 320.683,Z 495.361,A -85,B 0,C 180,E1 -15395.026,E2 -15395.026} C_VEL
LIN {X 0,Y 320.949,Z 492.586,A -85,B 0,C 180,E1 -15396.914,E2 -15396.914} C_VEL
LIN {X 0,Y 321.647,Z 488.759,A -85,B 0,C 180,E1 -15398.795,E2 -15398.795} C_VEL
LIN {X 0,Y 322.605,Z 483.783,A -85,B 0,C 180,E1 -15400.668,E2 -15400.668} C_VEL
LIN {X 0,Y 323.464,Z 477.547,A -85,B 0,C 180,E1 -15402.546,E2 -15402.546} C_VEL
LIN {X 0,Y 324.6,Z 469.765,A -85,B 0,C 180,E1 -15404.414,E2 -15404.414} C_VEL
LIN {X 0,Y 325.771,Z 461.782,A -85,B 0,C 180,E1 -15405.962,E2 -15405.962} C_VEL
LIN {X 0,Y 326.82,Z 453.074,A -85,B 0,C 180,E1 -15407.356,E2 -15407.356} C_VEL
LIN {X 0,Y 327.926,Z 442.263,A -85,B 0,C 180,E1 -15408.749,E2 -15408.749} C_VEL
LIN {X 0,Y 328.995,Z 431.005,A -85,B 0,C 180,E1 -15409.886,E2 -15409.886} C_VEL
LIN {X 0,Y 329.747,Z 419.696,A -85,B 0,C 180,E1 -15410.776,E2 -15410.776} C_VEL
LIN {X 0,Y 329.935,Z 411.988,A -85,B 0,C 180,E1 -15411.26,E2 -15411.26} C_VEL
LIN {X 0,Y 326.369,Z 400.11,A -85,B 0,C 180,E1 -15412.105,E2 -15412.105} C_VEL
LIN {X 0,Y 323.367,Z 391.681,A -85,B 0,C 180,E1 -15412.634,E2 -15412.634} C_VEL
LIN {X 0,Y 323.171,Z 382.763,A -85,B 0,C 180,E1 -15416.344,E2 -15416.344} C_VEL
LIN {X 0,Y 323.197,Z 373.035,A -85,B 0,C 180,E1 -15420.727,E2 -15420.727} C_VEL
LIN {X 0,Y 323.482,Z 363.677,A -85,B 0,C 180,E1 -15425.147,E2 -15425.147} C_VEL
LIN {X 0,Y 323.23,Z 358.952,A -85,B 0,C 180,E1 -15427.498,E2 -15427.498} C_VEL
LIN {X 0,Y 322.289,Z 353.393,A -85,B 0,C 180,E1 -15430.25,E2 -15430.25} C_VEL
LIN {X 0,Y 320.825,Z 346.444,A -85,B 0,C 180,E1 -15433.705,E2 -15433.705} C_VEL
LIN {X 0,Y 319.567,Z 340.992,A -85,B 0,C 180,E1 -15436.406,E2 -15436.406} C_VEL
LIN {X 0,Y 319.594,Z 340.987,A -85,B 0,C 180,E1 -15440.317,E2 -15440.317} C_VEL
LIN {X 0,Y 319.581,Z 340.987,A -85,B 0,C 180,E1 -15442.358,E2 -15442.358} C_VEL
LIN {X 0,Y 318.852,Z 341.081,A -85,B 0,C 180,E1 -15443.41,E2 -15443.41} C_VEL
LIN {X 0,Y 315.97,Z 341.439,A -85,B 0,C 180,E1 -15445.123,E2 -15445.123} C_VEL
LIN {X 0,Y 313.569,Z 341.735,A -85,B 0,C 180,E1 -15446.51,E2 -15446.51} C_VEL
LIN {X 0,Y 312.549,Z 341.862,A -85,B 0,C 180,E1 -15447.585,E2 -15447.585} C_VEL
LIN {X 0,Y 312.47,Z 341.871,A -85,B 0,C 180,E1 -15447.949,E2 -15447.949} C_VEL
LIN {X 0,Y 312.555,Z 341.865,A -85,B 0,C 180,E1 -15451.822,E2 -15451.822} C_VEL
LIN {X 0,Y 312.575,Z 341.861,A -85,B 0,C 180,E1 -15454.709,E2 -15454.709} C_VEL
LIN {X 0,Y 312.599,Z 341.849,A -85,B 0,C 180,E1 -15457.529,E2 -15457.529} C_VEL
LIN {X 0,Y 312.623,Z 341.846,A -85,B 0,C 180,E1 -15461.655,E2 -15461.655} C_VEL
LIN {X 0,Y 312.672,Z 341.836,A -85,B 0,C 180,E1 -15465.685,E2 -15465.685} C_VEL
LIN {X 0,Y 312.682,Z 341.84,A -85,B 0,C 180,E1 -15469.641,E2 -15469.641} C_VEL
LIN {X 0,Y 312.849,Z 341.827,A -85,B 0,C 180,E1 -15472.253,E2 -15472.253} C_VEL
LIN {X 0,Y 312.693,Z 341.837,A -85,B 0,C 180,E1 -15474.841,E2 -15474.841} C_VEL
LIN {X 0,Y 312.966,Z 341.813,A -85,B 0,C 180,E1 -15478.713,E2 -15478.713} C_VEL
LIN {X 0,Y 312.972,Z 341.8,A -85,B 0,C 180,E1 -15481.286,E2 -15481.286} C_VEL
LIN {X 0,Y 312.696,Z 341.848,A -85,B 0,C 180,E1 -15483.866,E2 -15483.866} C_VEL
LIN {X 0,Y 312.89,Z 341.821,A -85,B 0,C 180,E1 -15486.448,E2 -15486.448} C_VEL
LIN {X 0,Y 312.765,Z 341.838,A -85,B 0,C 180,E1 -15489.049,E2 -15489.049} C_VEL
LIN {X 0,Y 312.614,Z 341.857,A -85,B 0,C 180,E1 -15492.991,E2 -15492.991} C_VEL
LIN {X 0,Y 312.616,Z 341.858,A -85,B 0,C 180,E1 -15495.65,E2 -15495.65} C_VEL
LIN {X 0,Y 312.613,Z 341.857,A -85,B 0,C 180,E1 -15499.707,E2 -15499.707} C_VEL
LIN {X 0,Y 312.579,Z 341.862,A -85,B 0,C 180,E1 -15502.814,E2 -15502.814} C_VEL
LIN {X 0,Y 312.533,Z 341.865,A -85,B 0,C 180,E1 -15506.727,E2 -15506.727} C_VEL
LIN {X 0,Y 312.561,Z 341.962,A -85,B 0,C 180,E1 -15507.085,E2 -15507.085} C_VEL
LIN {X 0,Y 314.635,Z 349.652,A -85,B 0,C 180,E1 -15510.913,E2 -15510.913} C_VEL
LIN {X 0,Y 317.151,Z 358.406,A -85,B 0,C 180,E1 -15514.931,E2 -15514.931} C_VEL
LIN {X 0,Y 319.711,Z 367.626,A -85,B 0,C 180,E1 -15518.792,E2 -15518.792} C_VEL
LIN {X 0,Y 322.372,Z 377.305,A -85,B 0,C 180,E1 -15522.518,E2 -15522.518} C_VEL
LIN {X 0,Y 325.452,Z 387.84,A -85,B 0,C 180,E1 -15526.294,E2 -15526.294} C_VEL
LIN {X 0,Y 328.049,Z 397.914,A -85,B 0,C 180,E1 -15529.609,E2 -15529.609} C_VEL
LIN {X 0,Y 325.486,Z 408.354,A -85,B 0,C 180,E1 -15532.417,E2 -15532.417} C_VEL
LIN {X 0,Y 324.287,Z 413.536,A -85,B 0,C 180,E1 -15533.748,E2 -15533.748} C_VEL
LIN {X 0,Y 327.595,Z 436.013,A -85,B 0,C 180,E1 -15534.828,E2 -15534.828} C_VEL
LIN {X 0,Y 329.882,Z 452.918,A -85,B 0,C 180,E1 -15535.865,E2 -15535.865} C_VEL
LIN {X 0,Y 331.49,Z 468.469,A -85,B 0,C 180,E1 -15537.007,E2 -15537.007} C_VEL
LIN {X 0,Y 329.398,Z 483.724,A -85,B 0,C 180,E1 -15538.13,E2 -15538.13} C_VEL
LIN {X 0,Y 326.891,Z 498.973,A -85,B 0,C 180,E1 -15539.52,E2 -15539.52} C_VEL
LIN {X 0,Y 324.599,Z 512.5,A -85,B 0,C 180,E1 -15541.028,E2 -15541.028} C_VEL
LIN {X 0,Y 322.102,Z 525.409,A -85,B 0,C 180,E1 -15542.733,E2 -15542.733} C_VEL
LIN {X 0,Y 319.684,Z 537.676,A -85,B 0,C 180,E1 -15544.658,E2 -15544.658} C_VEL
LIN {X 0,Y 317.425,Z 549.467,A -85,B 0,C 180,E1 -15546.863,E2 -15546.863} C_VEL
LIN {X 0,Y 315.353,Z 560.715,A -85,B 0,C 180,E1 -15549.392,E2 -15549.392} C_VEL
LIN {X 0,Y 313.749,Z 570.535,A -85,B 0,C 180,E1 -15552.065,E2 -15552.065} C_VEL
LIN {X 0,Y 312.521,Z 579.284,A -85,B 0,C 180,E1 -15555.001,E2 -15555.001} C_VEL
LIN {X 0,Y 311.885,Z 585.596,A -85,B 0,C 180,E1 -15557.642,E2 -15557.642} C_VEL
LIN {X 0,Y 311.578,Z 590.539,A -85,B 0,C 180,E1 -15560.264,E2 -15560.264} C_VEL
LIN {X 0,Y 311.556,Z 594.434,A -85,B 0,C 180,E1 -15562.993,E2 -15562.993} C_VEL
LIN {X 0,Y 311.693,Z 597.317,A -85,B 0,C 180,E1 -15566.125,E2 -15566.125} C_VEL
LIN {X 0,Y 311.641,Z 598.412,A -85,B 0,C 180,E1 -15568.711,E2 -15568.711} C_VEL
LIN {X 0,Y 311.639,Z 598.387,A -85,B 0,C 180,E1 -15571.295,E2 -15571.295} C_VEL
LIN {X 0,Y 311.709,Z 597.306,A -85,B 0,C 180,E1 -15573.882,E2 -15573.882} C_VEL
LIN {X 0,Y 311.574,Z 594.414,A -85,B 0,C 180,E1 -15577.033,E2 -15577.033} C_VEL
LIN {X 0,Y 311.531,Z 590.618,A -85,B 0,C 180,E1 -15579.744,E2 -15579.744} C_VEL
LIN {X 0,Y 311.864,Z 585.871,A -85,B 0,C 180,E1 -15582.365,E2 -15582.365} C_VEL
LIN {X 0,Y 312.501,Z 579.88,A -85,B 0,C 180,E1 -15584.991,E2 -15584.991} C_VEL
LIN {X 0,Y 313.549,Z 572.641,A -85,B 0,C 180,E1 -15587.616,E2 -15587.616} C_VEL
LIN {X 0,Y 314.94,Z 564.659,A -85,B 0,C 180,E1 -15590.075,E2 -15590.075} C_VEL
LIN {X 0,Y 317.164,Z 554.047,A -85,B 0,C 180,E1 -15592.819,E2 -15592.819} C_VEL
LIN {X 0,Y 319.881,Z 542.288,A -85,B 0,C 180,E1 -15595.37,E2 -15595.37} C_VEL
LIN {X 0,Y 322.774,Z 530.333,A -85,B 0,C 180,E1 -15597.564,E2 -15597.564} C_VEL
LIN {X 0,Y 326.247,Z 516.572,A -85,B 0,C 180,E1 -15599.703,E2 -15599.703} C_VEL
LIN {X 0,Y 329.608,Z 503.092,A -85,B 0,C 180,E1 -15601.473,E2 -15601.473} C_VEL
LIN {X 0,Y 333.103,Z 488.53,A -85,B 0,C 180,E1 -15603.091,E2 -15603.091} C_VEL
LIN {X 0,Y 336.968,Z 471.551,A -85,B 0,C 180,E1 -15604.643,E2 -15604.643} C_VEL
LIN {X 0,Y 337.624,Z 459.154,A -85,B 0,C 180,E1 -15605.919,E2 -15605.919} C_VEL
LIN {X 0,Y 338.236,Z 444.989,A -85,B 0,C 180,E1 -15607.238,E2 -15607.238} C_VEL
LIN {X 0,Y 337.517,Z 431.155,A -85,B 0,C 180,E1 -15608.692,E2 -15608.692} C_VEL
LIN {X 0,Y 336.147,Z 419.965,A -85,B 0,C 180,E1 -15610.051,E2 -15610.051} C_VEL
LIN {X 0,Y 334.687,Z 411.169,A -85,B 0,C 180,E1 -15611.324,E2 -15611.324} C_VEL
LIN {X 0,Y 331.215,Z 404.418,A -85,B 0,C 180,E1 -15613.468,E2 -15613.468} C_VEL
LIN {X 0,Y 329.863,Z 400.855,A -85,B 0,C 180,E1 -15616.422,E2 -15616.422} C_VEL
LIN {X 0,Y 328.961,Z 399.064,A -85,B 0,C 180,E1 -15618.526,E2 -15618.526} C_VEL
LIN {X 0,Y 328.088,Z 398.069,A -85,B 0,C 180,E1 -15620.461,E2 -15620.461} C_VEL
LIN {X 0,Y 326.866,Z 397.687,A -85,B 0,C 180,E1 -15622.846,E2 -15622.846} C_VEL
LIN {X 0,Y 327.705,Z 400.325,A -85,B 0,C 180,E1 -15624.617,E2 -15624.617} C_VEL
LIN {X 0,Y 328.555,Z 401.408,A -85,B 0,C 180,E1 -15625.485,E2 -15625.485} C_VEL
LIN {X 0,Y 329.18,Z 403.588,A -85,B 0,C 180,E1 -15626.376,E2 -15626.376} C_VEL
LIN {X 0,Y 330.413,Z 406.073,A -85,B 0,C 180,E1 -15627.515,E2 -15627.515} C_VEL
LIN {X 0,Y 332.313,Z 410.636,A -85,B 0,C 180,E1 -15629.146,E2 -15629.146} C_VEL
LIN {X 0,Y 334.33,Z 415.784,A -85,B 0,C 180,E1 -15630.719,E2 -15630.719} C_VEL
LIN {X 0,Y 336.748,Z 423.372,A -85,B 0,C 180,E1 -15632.669,E2 -15632.669} C_VEL
LIN {X 0,Y 338.605,Z 432.128,A -85,B 0,C 180,E1 -15634.563,E2 -15634.563} C_VEL
LIN {X 0,Y 338.696,Z 433.252,A -85,B 0,C 180,E1 -15634.771,E2 -15634.771} C_VEL
LIN {X 0,Y 335.231,Z 446.376,A -85,B 0,C 180,E1 -15636.363,E2 -15636.363} C_VEL
LIN {X 0,Y 332.203,Z 457.202,A -85,B 0,C 180,E1 -15637.944,E2 -15637.944} C_VEL
LIN {X 0,Y 328.764,Z 468.706,A -85,B 0,C 180,E1 -15640,E2 -15640} C_VEL
LIN {X 0,Y 326.201,Z 476.815,A -85,B 0,C 180,E1 -15641.754,E2 -15641.754} C_VEL
LIN {X 0,Y 323.458,Z 485.123,A -85,B 0,C 180,E1 -15643.918,E2 -15643.918} C_VEL
LIN {X 0,Y 321.155,Z 491.637,A -85,B 0,C 180,E1 -15646.072,E2 -15646.072} C_VEL
LIN {X 0,Y 319.357,Z 496.157,A -85,B 0,C 180,E1 -15647.933,E2 -15647.933} C_VEL
LIN {X 0,Y 317.845,Z 499.67,A -85,B 0,C 180,E1 -15649.812,E2 -15649.812} C_VEL
LIN {X 0,Y 317.019,Z 501.5,A -85,B 0,C 180,E1 -15651.073,E2 -15651.073} C_VEL
LIN {X 0,Y 315.777,Z 503.868,A -85,B 0,C 180,E1 -15653.611,E2 -15653.611} C_VEL
LIN {X 0,Y 314.72,Z 504.748,A -85,B 0,C 180,E1 -15656.159,E2 -15656.159} C_VEL
LIN {X 0,Y 314.258,Z 504.61,A -85,B 0,C 180,E1 -15657.437,E2 -15657.437} C_VEL
LIN {X 0,Y 313.93,Z 504.053,A -85,B 0,C 180,E1 -15658.718,E2 -15658.718} C_VEL
LIN {X 0,Y 313.647,Z 503.075,A -85,B 0,C 180,E1 -15660.001,E2 -15660.001} C_VEL
LIN {X 0,Y 313.516,Z 501.678,A -85,B 0,C 180,E1 -15661.285,E2 -15661.285} C_VEL
LIN {X 0,Y 313.428,Z 498.813,A -85,B 0,C 180,E1 -15663.214,E2 -15663.214} C_VEL
LIN {X 0,Y 313.443,Z 494.989,A -85,B 0,C 180,E1 -15665.146,E2 -15665.146} C_VEL
LIN {X 0,Y 313.602,Z 490.116,A -85,B 0,C 180,E1 -15667.081,E2 -15667.081} C_VEL
LIN {X 0,Y 314.196,Z 484.075,A -85,B 0,C 180,E1 -15669.009,E2 -15669.009} C_VEL
LIN {X 0,Y 314.782,Z 475.564,A -85,B 0,C 180,E1 -15671.234,E2 -15671.234} C_VEL
LIN {X 0,Y 315.6,Z 466.425,A -85,B 0,C 180,E1 -15673.195,E2 -15673.195} C_VEL
LIN {X 0,Y 316.53,Z 455.598,A -85,B 0,C 180,E1 -15675.123,E2 -15675.123} C_VEL
LIN {X 0,Y 317.786,Z 443.61,A -85,B 0,C 180,E1 -15676.874,E2 -15676.874} C_VEL
LIN {X 0,Y 318.868,Z 431.114,A -85,B 0,C 180,E1 -15678.394,E2 -15678.394} C_VEL
LIN {X 0,Y 319.954,Z 417.586,A -85,B 0,C 180,E1 -15679.739,E2 -15679.739} C_VEL
LIN {X 0,Y 320.803,Z 408.128,A -85,B 0,C 180,E1 -15680.52,E2 -15680.52} C_VEL
LIN {X 0,Y 318.351,Z 395.901,A -85,B 0,C 180,E1 -15681.566,E2 -15681.566} C_VEL
LIN {X 0,Y 314.647,Z 379.951,A -85,B 0,C 180,E1 -15682.724,E2 -15682.724} C_VEL
LIN {X 0,Y 312.946,Z 373.311,A -85,B 0,C 180,E1 -15683.139,E2 -15683.139} C_VEL
LIN {X 0,Y 313.303,Z 366.447,A -85,B 0,C 180,E1 -15687.378,E2 -15687.378} C_VEL
LIN {X 0,Y 313.697,Z 360.684,A -85,B 0,C 180,E1 -15691.017,E2 -15691.017} C_VEL
LIN {X 0,Y 314.106,Z 354.882,A -85,B 0,C 180,E1 -15694.789,E2 -15694.789} C_VEL
LIN {X 0,Y 314.086,Z 351.371,A -85,B 0,C 180,E1 -15697.169,E2 -15697.169} C_VEL
LIN {X 0,Y 313.362,Z 346.61,A -85,B 0,C 180,E1 -15700.573,E2 -15700.573} C_VEL
LIN {X 0,Y 312.711,Z 342.812,A -85,B 0,C 180,E1 -15703.47,E2 -15703.47} C_VEL
LIN {X 0,Y 314.197,Z 349.201,A -85,B 0,C 180,E1 -15706.647,E2 -15706.647} C_VEL
LIN {X 0,Y 315.476,Z 355.343,A -85,B 0,C 180,E1 -15709.753,E2 -15709.753} C_VEL
LIN {X 0,Y 316.395,Z 360.474,A -85,B 0,C 180,E1 -15712.347,E2 -15712.347} C_VEL
LIN {X 0,Y 316.627,Z 365.308,A -85,B 0,C 180,E1 -15714.75,E2 -15714.75} C_VEL
LIN {X 0,Y 316.411,Z 373.429,A -85,B 0,C 180,E1 -15718.532,E2 -15718.532} C_VEL
LIN {X 0,Y 316.382,Z 383.114,A -85,B 0,C 180,E1 -15722.944,E2 -15722.944} C_VEL
LIN {X 0,Y 316.542,Z 392.249,A -85,B 0,C 180,E1 -15726.788,E2 -15726.788} C_VEL
LIN {X 0,Y 316.575,Z 392.737,A -85,B 0,C 180,E1 -15726.989,E2 -15726.989} C_VEL
LIN {X 0,Y 321.329,Z 406.421,A -85,B 0,C 180,E1 -15727.878,E2 -15727.878} C_VEL
LIN {X 0,Y 323.462,Z 414.454,A -85,B 0,C 180,E1 -15728.489,E2 -15728.489} C_VEL
LIN {X 0,Y 322.844,Z 425.843,A -85,B 0,C 180,E1 -15729.268,E2 -15729.268} C_VEL
LIN {X 0,Y 321.959,Z 437.114,A -85,B 0,C 180,E1 -15730.287,E2 -15730.287} C_VEL
LIN {X 0,Y 321.041,Z 446.316,A -85,B 0,C 180,E1 -15731.325,E2 -15731.325} C_VEL
LIN {X 0,Y 319.614,Z 457.521,A -85,B 0,C 180,E1 -15732.893,E2 -15732.893} C_VEL
LIN {X 0,Y 318.604,Z 465.658,A -85,B 0,C 180,E1 -15734.32,E2 -15734.32} C_VEL
LIN {X 0,Y 317.467,Z 473.173,A -85,B 0,C 180,E1 -15735.903,E2 -15735.903} C_VEL
LIN {X 0,Y 316.326,Z 480.579,A -85,B 0,C 180,E1 -15737.845,E2 -15737.845} C_VEL
LIN {X 0,Y 315.463,Z 486.31,A -85,B 0,C 180,E1 -15739.731,E2 -15739.731} C_VEL
LIN {X 0,Y 314.366,Z 490.981,A -85,B 0,C 180,E1 -15741.642,E2 -15741.642} C_VEL
LIN {X 0,Y 313.784,Z 494.509,A -85,B 0,C 180,E1 -15743.567,E2 -15743.567} C_VEL
LIN {X 0,Y 313.679,Z 496.294,A -85,B 0,C 180,E1 -15744.855,E2 -15744.855} C_VEL
LIN {X 0,Y 313.422,Z 497.684,A -85,B 0,C 180,E1 -15746.14,E2 -15746.14} C_VEL
LIN {X 0,Y 313.066,Z 499.267,A -85,B 0,C 180,E1 -15748.711,E2 -15748.711} C_VEL
LIN {X 0,Y 313.038,Z 499.496,A -85,B 0,C 180,E1 -15749.997,E2 -15749.997} C_VEL
LIN {X 0,Y 313.161,Z 498.735,A -85,B 0,C 180,E1 -15752.569,E2 -15752.569} C_VEL
LIN {X 0,Y 313.432,Z 497.775,A -85,B 0,C 180,E1 -15753.854,E2 -15753.854} C_VEL
LIN {X 0,Y 313.695,Z 496.437,A -85,B 0,C 180,E1 -15755.138,E2 -15755.138} C_VEL
LIN {X 0,Y 313.981,Z 493.662,A -85,B 0,C 180,E1 -15757.068,E2 -15757.068} C_VEL
LIN {X 0,Y 314.713,Z 489.833,A -85,B 0,C 180,E1 -15758.99,E2 -15758.99} C_VEL
LIN {X 0,Y 315.715,Z 484.855,A -85,B 0,C 180,E1 -15760.904,E2 -15760.904} C_VEL
LIN {X 0,Y 316.619,Z 478.618,A -85,B 0,C 180,E1 -15762.821,E2 -15762.821} C_VEL
LIN {X 0,Y 317.808,Z 470.835,A -85,B 0,C 180,E1 -15764.729,E2 -15764.729} C_VEL
LIN {X 0,Y 319.027,Z 462.849,A -85,B 0,C 180,E1 -15766.309,E2 -15766.309} C_VEL
LIN {X 0,Y 320.127,Z 454.137,A -85,B 0,C 180,E1 -15767.731,E2 -15767.731} C_VEL
LIN {X 0,Y 321.285,Z 443.32,A -85,B 0,C 180,E1 -15769.151,E2 -15769.151} C_VEL
LIN {X 0,Y 322.304,Z 433.041,A -85,B 0,C 180,E1 -15770.219,E2 -15770.219} C_VEL
LIN {X 0,Y 323.117,Z 421.734,A -85,B 0,C 180,E1 -15771.146,E2 -15771.146} C_VEL
LIN {X 0,Y 323.367,Z 413.587,A -85,B 0,C 180,E1 -15771.679,E2 -15771.679} C_VEL
LIN {X 0,Y 319.686,Z 401.407,A -85,B 0,C 180,E1 -15772.581,E2 -15772.581} C_VEL
LIN {X 0,Y 316.582,Z 392.75,A -85,B 0,C 180,E1 -15773.128,E2 -15773.128} C_VEL
LIN {X 0,Y 316.391,Z 383.415,A -85,B 0,C 180,E1 -15777.059,E2 -15777.059} C_VEL
LIN {X 0,Y 316.465,Z 373.709,A -85,B 0,C 180,E1 -15781.454,E2 -15781.454} C_VEL
LIN {X 0,Y 316.723,Z 365.761,A -85,B 0,C 180,E1 -15785.23,E2 -15785.23} C_VEL
LIN {X 0,Y 316.67,Z 362.318,A -85,B 0,C 180,E1 -15786.968,E2 -15786.968} C_VEL
LIN {X 0,Y 315.562,Z 355.672,A -85,B 0,C 180,E1 -15790.226,E2 -15790.226} C_VEL
LIN {X 0,Y 314.331,Z 349.604,A -85,B 0,C 180,E1 -15793.357,E2 -15793.357} C_VEL
LIN {X 0,Y 312.55,Z 341.867,A -85,B 0,C 180,E1 -15797.14,E2 -15797.14} C_VEL
LIN {X 0,Y 312.523,Z 341.869,A -85,B 0,C 180,E1 -15800.974,E2 -15800.974} C_VEL
LIN {X 0,Y 312.516,Z 341.865,A -85,B 0,C 180,E1 -15804.218,E2 -15804.218} C_VEL
LIN {X 0,Y 312.47,Z 341.871,A -85,B 0,C 180,E1 -15807.949,E2 -15807.949} C_VEL
LIN {X 0,Y 311.808,Z 341.958,A -85,B 0,C 180,E1 -15809.025,E2 -15809.025} C_VEL
LIN {X 0,Y 308.957,Z 342.309,A -85,B 0,C 180,E1 -15810.776,E2 -15810.776} C_VEL
LIN {X 0,Y 306.565,Z 342.611,A -85,B 0,C 180,E1 -15812.197,E2 -15812.197} C_VEL
LIN {X 0,Y 305.58,Z 342.725,A -85,B 0,C 180,E1 -15813.297,E2 -15813.297} C_VEL
LIN {X 0,Y 305.522,Z 342.731,A -85,B 0,C 180,E1 -15813.669,E2 -15813.669} C_VEL
LIN {X 0,Y 305.517,Z 342.731,A -85,B 0,C 180,E1 -15816.979,E2 -15816.979} C_VEL
LIN {X 0,Y 305.58,Z 342.723,A -85,B 0,C 180,E1 -15821.216,E2 -15821.216} C_VEL
LIN {X 0,Y 305.627,Z 342.714,A -85,B 0,C 180,E1 -15825.347,E2 -15825.347} C_VEL
LIN {X 0,Y 305.619,Z 342.722,A -85,B 0,C 180,E1 -15829.399,E2 -15829.399} C_VEL
LIN {X 0,Y 305.79,Z 342.703,A -85,B 0,C 180,E1 -15832.073,E2 -15832.073} C_VEL
LIN {X 0,Y 305.665,Z 342.713,A -85,B 0,C 180,E1 -15834.723,E2 -15834.723} C_VEL
LIN {X 0,Y 305.933,Z 342.689,A -85,B 0,C 180,E1 -15838.683,E2 -15838.683} C_VEL
LIN {X 0,Y 305.939,Z 342.675,A -85,B 0,C 180,E1 -15841.316,E2 -15841.316} C_VEL
LIN {X 0,Y 305.676,Z 342.721,A -85,B 0,C 180,E1 -15845.276,E2 -15845.276} C_VEL
LIN {X 0,Y 305.79,Z 342.709,A -85,B 0,C 180,E1 -15847.926,E2 -15847.926} C_VEL
LIN {X 0,Y 305.583,Z 342.734,A -85,B 0,C 180,E1 -15851.945,E2 -15851.945} C_VEL
LIN {X 0,Y 305.615,Z 342.729,A -85,B 0,C 180,E1 -15855.035,E2 -15855.035} C_VEL
LIN {X 0,Y 305.592,Z 342.734,A -85,B 0,C 180,E1 -15859.466,E2 -15859.466} C_VEL
LIN {X 0,Y 305.533,Z 342.738,A -85,B 0,C 180,E1 -15863.071,E2 -15863.071} C_VEL
LIN {X 0,Y 305.543,Z 342.831,A -85,B 0,C 180,E1 -15866.003,E2 -15866.003} C_VEL
LIN {X 0,Y 307.715,Z 350.909,A -85,B 0,C 180,E1 -15870.163,E2 -15870.163} C_VEL
LIN {X 0,Y 310.285,Z 360.115,A -85,B 0,C 180,E1 -15874.489,E2 -15874.489} C_VEL
LIN {X 0,Y 312.648,Z 368.555,A -85,B 0,C 180,E1 -15878.123,E2 -15878.123} C_VEL
LIN {X 0,Y 315.312,Z 378.238,A -85,B 0,C 180,E1 -15881.964,E2 -15881.964} C_VEL
LIN {X 0,Y 318.357,Z 388.788,A -85,B 0,C 180,E1 -15885.845,E2 -15885.845} C_VEL
LIN {X 0,Y 321.021,Z 398.988,A -85,B 0,C 180,E1 -15889.292,E2 -15889.292} C_VEL
LIN {X 0,Y 321.056,Z 400.138,A -85,B 0,C 180,E1 -15889.641,E2 -15889.641} C_VEL
LIN {X 0,Y 317.673,Z 413.215,A -85,B 0,C 180,E1 -15893.172,E2 -15893.172} C_VEL
LIN {X 0,Y 320.95,Z 436.265,A -85,B 0,C 180,E1 -15894.312,E2 -15894.312} C_VEL
LIN {X 0,Y 323.153,Z 452.675,A -85,B 0,C 180,E1 -15895.353,E2 -15895.353} C_VEL
LIN {X 0,Y 324.734,Z 468.865,A -85,B 0,C 180,E1 -15896.581,E2 -15896.581} C_VEL
LIN {X 0,Y 322.634,Z 484.157,A -85,B 0,C 180,E1 -15897.749,E2 -15897.749} C_VEL
LIN {X 0,Y 320.011,Z 499.757,A -85,B 0,C 180,E1 -15899.225,E2 -15899.225} C_VEL
LIN {X 0,Y 317.481,Z 513.836,A -85,B 0,C 180,E1 -15900.86,E2 -15900.86} C_VEL
LIN {X 0,Y 314.764,Z 527.474,A -85,B 0,C 180,E1 -15902.764,E2 -15902.764} C_VEL
LIN {X 0,Y 312.431,Z 539.093,A -85,B 0,C 180,E1 -15904.702,E2 -15904.702} C_VEL
LIN {X 0,Y 310.115,Z 550.678,A -85,B 0,C 180,E1 -15906.992,E2 -15906.992} C_VEL
LIN {X 0,Y 308.108,Z 561.446,A -85,B 0,C 180,E1 -15909.546,E2 -15909.546} C_VEL
LIN {X 0,Y 306.57,Z 571.094,A -85,B 0,C 180,E1 -15912.321,E2 -15912.321} C_VEL
LIN {X 0,Y 305.437,Z 578.989,A -85,B 0,C 180,E1 -15915.105,E2 -15915.105} C_VEL
LIN {X 0,Y 304.754,Z 585.613,A -85,B 0,C 180,E1 -15918.025,E2 -15918.025} C_VEL
LIN {X 0,Y 304.517,Z 590.339,A -85,B 0,C 180,E1 -15920.706,E2 -15920.706} C_VEL
LIN {X 0,Y 304.519,Z 593.819,A -85,B 0,C 180,E1 -15923.377,E2 -15923.377} C_VEL
LIN {X 0,Y 304.665,Z 596.176,A -85,B 0,C 180,E1 -15926.035,E2 -15926.035} C_VEL
LIN {X 0,Y 304.627,Z 597.292,A -85,B 0,C 180,E1 -15928.681,E2 -15928.681} C_VEL
LIN {X 0,Y 304.617,Z 597.313,A -85,B 0,C 180,E1 -15931.325,E2 -15931.325} C_VEL
LIN {X 0,Y 304.682,Z 596.243,A -85,B 0,C 180,E1 -15933.971,E2 -15933.971} C_VEL
LIN {X 0,Y 304.515,Z 593.521,A -85,B 0,C 180,E1 -15937.068,E2 -15937.068} C_VEL
LIN {X 0,Y 304.472,Z 589.632,A -85,B 0,C 180,E1 -15939.972,E2 -15939.972} C_VEL
LIN {X 0,Y 304.816,Z 584.929,A -85,B 0,C 180,E1 -15942.655,E2 -15942.655} C_VEL
LIN {X 0,Y 305.712,Z 577.332,A -85,B 0,C 180,E1 -15946.017,E2 -15946.017} C_VEL
LIN {X 0,Y 307.159,Z 568.841,A -85,B 0,C 180,E1 -15949.032,E2 -15949.032} C_VEL
LIN {X 0,Y 309.288,Z 558.61,A -85,B 0,C 180,E1 -15952.023,E2 -15952.023} C_VEL
LIN {X 0,Y 311.84,Z 547.867,A -85,B 0,C 180,E1 -15954.644,E2 -15954.644} C_VEL
LIN {X 0,Y 315.105,Z 535.375,A -85,B 0,C 180,E1 -15957.211,E2 -15957.211} C_VEL
LIN {X 0,Y 318.423,Z 522.708,A -85,B 0,C 180,E1 -15959.415,E2 -15959.415} C_VEL
LIN {X 0,Y 322.381,Z 508.097,A -85,B 0,C 180,E1 -15961.55,E2 -15961.55} C_VEL
LIN {X 0,Y 326.22,Z 493.557,A -85,B 0,C 180,E1 -15963.326,E2 -15963.326} C_VEL
LIN {X 0,Y 330.171,Z 478.057,A -85,B 0,C 180,E1 -15964.897,E2 -15964.897} C_VEL
LIN {X 0,Y 331.35,Z 472.968,A -85,B 0,C 180,E1 -15965.363,E2 -15965.363} C_VEL
LIN {X 0,Y 332.531,Z 458.792,A -85,B 0,C 180,E1 -15966.877,E2 -15966.877} C_VEL
LIN {X 0,Y 333.347,Z 446.095,A -85,B 0,C 180,E1 -15968.133,E2 -15968.133} C_VEL
LIN {X 0,Y 333.03,Z 433.922,A -85,B 0,C 180,E1 -15969.519,E2 -15969.519} C_VEL
LIN {X 0,Y 332.238,Z 424.008,A -85,B 0,C 180,E1 -15970.797,E2 -15970.797} C_VEL
LIN {X 0,Y 331.31,Z 416.523,A -85,B 0,C 180,E1 -15971.912,E2 -15971.912} C_VEL
LIN {X 0,Y 328.283,Z 410.463,A -85,B 0,C 180,E1 -15973.941,E2 -15973.941} C_VEL
LIN {X 0,Y 325.582,Z 406.62,A -85,B 0,C 180,E1 -15976.311,E2 -15976.311} C_VEL
LIN {X 0,Y 324.555,Z 404.96,A -85,B 0,C 180,E1 -15977.835,E2 -15977.835} C_VEL
LIN {X 0,Y 323.99,Z 404.031,A -85,B 0,C 180,E1 -15979.402,E2 -15979.402} C_VEL
LIN {X 0,Y 323.987,Z 403.87,A -85,B 0,C 180,E1 -15981.348,E2 -15981.348} C_VEL
LIN {X 0,Y 324.437,Z 404.279,A -85,B 0,C 180,E1 -15982.661,E2 -15982.661} C_VEL
LIN {X 0,Y 325.013,Z 406.626,A -85,B 0,C 180,E1 -15984.279,E2 -15984.279} C_VEL
LIN {X 0,Y 325.63,Z 407.61,A -85,B 0,C 180,E1 -15985.103,E2 -15985.103} C_VEL
LIN {X 0,Y 326.088,Z 409.495,A -85,B 0,C 180,E1 -15985.92,E2 -15985.92} C_VEL
LIN {X 0,Y 327.01,Z 411.472,A -85,B 0,C 180,E1 -15986.951,E2 -15986.951} C_VEL
LIN {X 0,Y 329.43,Z 418.304,A -85,B 0,C 180,E1 -15989.464,E2 -15989.464} C_VEL
LIN {X 0,Y 331.714,Z 426.351,A -85,B 0,C 180,E1 -15991.77,E2 -15991.77} C_VEL
LIN {X 0,Y 333.086,Z 433.063,A -85,B 0,C 180,E1 -15993.375,E2 -15993.375} C_VEL
LIN {X 0,Y 333.49,Z 435.621,A -85,B 0,C 180,E1 -15993.943,E2 -15993.943} C_VEL
LIN {X 0,Y 333.416,Z 436.839,A -85,B 0,C 180,E1 -15994.147,E2 -15994.147} C_VEL
LIN {X 0,Y 329.388,Z 450.59,A -85,B 0,C 180,E1 -15995.917,E2 -15995.917} C_VEL
LIN {X 0,Y 325.677,Z 462.505,A -85,B 0,C 180,E1 -15997.813,E2 -15997.813} C_VEL
LIN {X 0,Y 322.632,Z 471.848,A -85,B 0,C 180,E1 -15999.603,E2 -15999.603} C_VEL
LIN {X 0,Y 319.453,Z 480.998,A -85,B 0,C 180,E1 -16001.73,E2 -16001.73} C_VEL
LIN {X 0,Y 316.657,Z 488.524,A -85,B 0,C 180,E1 -16003.894,E2 -16003.894} C_VEL
LIN {X 0,Y 314.59,Z 493.808,A -85,B 0,C 180,E1 -16005.775,E2 -16005.775} C_VEL
LIN {X 0,Y 312.122,Z 499.377,A -85,B 0,C 180,E1 -16008.308,E2 -16008.308} C_VEL
LIN {X 0,Y 311.111,Z 501.503,A -85,B 0,C 180,E1 -16009.589,E2 -16009.589} C_VEL
LIN {X 0,Y 309.486,Z 504.508,A -85,B 0,C 180,E1 -16012.169,E2 -16012.169} C_VEL
LIN {X 0,Y 308.91,Z 505.41,A -85,B 0,C 180,E1 -16013.469,E2 -16013.469} C_VEL
LIN {X 0,Y 307.785,Z 506.12,A -85,B 0,C 180,E1 -16016.073,E2 -16016.073} C_VEL
LIN {X 0,Y 307.3,Z 505.898,A -85,B 0,C 180,E1 -16017.379,E2 -16017.379} C_VEL
LIN {X 0,Y 306.942,Z 505.24,A -85,B 0,C 180,E1 -16018.689,E2 -16018.689} C_VEL
LIN {X 0,Y 306.638,Z 504.184,A -85,B 0,C 180,E1 -16020.001,E2 -16020.001} C_VEL
LIN {X 0,Y 306.507,Z 502.712,A -85,B 0,C 180,E1 -16021.314,E2 -16021.314} C_VEL
LIN {X 0,Y 306.402,Z 499.732,A -85,B 0,C 180,E1 -16023.288,E2 -16023.288} C_VEL
LIN {X 0,Y 306.406,Z 495.774,A -85,B 0,C 180,E1 -16025.265,E2 -16025.265} C_VEL
LIN {X 0,Y 306.596,Z 490.773,A -85,B 0,C 180,E1 -16027.243,E2 -16027.243} C_VEL
LIN {X 0,Y 307.216,Z 484.623,A -85,B 0,C 180,E1 -16029.215,E2 -16029.215} C_VEL
LIN {X 0,Y 307.841,Z 475.811,A -85,B 0,C 180,E1 -16031.523,E2 -16031.523} C_VEL
LIN {X 0,Y 308.678,Z 466.648,A -85,B 0,C 180,E1 -16033.496,E2 -16033.496} C_VEL
LIN {X 0,Y 309.676,Z 455.601,A -85,B 0,C 180,E1 -16035.466,E2 -16035.466} C_VEL
LIN {X 0,Y 310.925,Z 443.457,A -85,B 0,C 180,E1 -16037.258,E2 -16037.258} C_VEL
LIN {X 0,Y 312.051,Z 430.741,A -85,B 0,C 180,E1 -16038.811,E2 -16038.811} C_VEL
LIN {X 0,Y 313.251,Z 417.074,A -85,B 0,C 180,E1 -16040.179,E2 -16040.179} C_VEL
LIN {X 0,Y 313.905,Z 408.429,A -85,B 0,C 180,E1 -16040.906,E2 -16040.906} C_VEL
LIN {X 0,Y 310.756,Z 393.58,A -85,B 0,C 180,E1 -16042.194,E2 -16042.194} C_VEL
LIN {X 0,Y 307.046,Z 378.064,A -85,B 0,C 180,E1 -16043.304,E2 -16043.304} C_VEL
LIN {X 0,Y 305.959,Z 373.685,A -85,B 0,C 180,E1 -16043.605,E2 -16043.605} C_VEL
LIN {X 0,Y 306.289,Z 367.746,A -85,B 0,C 180,E1 -16047.318,E2 -16047.318} C_VEL
LIN {X 0,Y 306.707,Z 361.927,A -85,B 0,C 180,E1 -16051.036,E2 -16051.036} C_VEL
LIN {X 0,Y 307.128,Z 356.084,A -85,B 0,C 180,E1 -16054.896,E2 -16054.896} C_VEL
LIN {X 0,Y 307.177,Z 353.292,A -85,B 0,C 180,E1 -16056.792,E2 -16056.792} C_VEL
LIN {X 0,Y 306.583,Z 348.929,A -85,B 0,C 180,E1 -16059.932,E2 -16059.932} C_VEL
LIN {X 0,Y 305.853,Z 344.729,A -85,B 0,C 180,E1 -16063.08,E2 -16063.08} C_VEL
LIN {X 0,Y 307.277,Z 350.348,A -85,B 0,C 180,E1 -16065.959,E2 -16065.959} C_VEL
LIN {X 0,Y 308.705,Z 357.364,A -85,B 0,C 180,E1 -16069.613,E2 -16069.613} C_VEL
LIN {X 0,Y 309.709,Z 363.282,A -85,B 0,C 180,E1 -16072.583,E2 -16072.583} C_VEL
LIN {X 0,Y 309.875,Z 367.644,A -85,B 0,C 180,E1 -16074.735,E2 -16074.735} C_VEL
LIN {X 0,Y 309.63,Z 375.712,A -85,B 0,C 180,E1 -16078.527,E2 -16078.527} C_VEL
LIN {X 0,Y 309.629,Z 385.554,A -85,B 0,C 180,E1 -16082.999,E2 -16082.999} C_VEL
LIN {X 0,Y 309.776,Z 393.769,A -85,B 0,C 180,E1 -16086.458,E2 -16086.458} C_VEL
LIN {X 0,Y 314.418,Z 407.068,A -85,B 0,C 180,E1 -16087.342,E2 -16087.342} C_VEL
LIN {X 0,Y 316.911,Z 416.154,A -85,B 0,C 180,E1 -16088.061,E2 -16088.061} C_VEL
LIN {X 0,Y 316.13,Z 428.489,A -85,B 0,C 180,E1 -16088.949,E2 -16088.949} C_VEL
LIN {X 0,Y 315.152,Z 440.323,A -85,B 0,C 180,E1 -16090.084,E2 -16090.084} C_VEL
LIN {X 0,Y 313.999,Z 451.051,A -85,B 0,C 180,E1 -16091.398,E2 -16091.398} C_VEL
LIN {X 0,Y 312.548,Z 461.453,A -85,B 0,C 180,E1 -16093,E2 -16093} C_VEL
LIN {X 0,Y 311.339,Z 469.896,A -85,B 0,C 180,E1 -16094.616,E2 -16094.616} C_VEL
LIN {X 0,Y 309.992,Z 478.11,A -85,B 0,C 180,E1 -16096.56,E2 -16096.56} C_VEL
LIN {X 0,Y 308.875,Z 485.59,A -85,B 0,C 180,E1 -16098.845,E2 -16098.845} C_VEL
LIN {X 0,Y 307.798,Z 490.644,A -85,B 0,C 180,E1 -16100.8,E2 -16100.8} C_VEL
LIN {X 0,Y 307.035,Z 494.538,A -85,B 0,C 180,E1 -16102.765,E2 -16102.765} C_VEL
LIN {X 0,Y 306.695,Z 497.371,A -85,B 0,C 180,E1 -16104.738,E2 -16104.738} C_VEL
LIN {X 0,Y 306.421,Z 498.761,A -85,B 0,C 180,E1 -16106.051,E2 -16106.051} C_VEL
LIN {X 0,Y 306.064,Z 500.342,A -85,B 0,C 180,E1 -16108.681,E2 -16108.681} C_VEL
LIN {X 0,Y 306.03,Z 500.571,A -85,B 0,C 180,E1 -16109.997,E2 -16109.997} C_VEL
LIN {X 0,Y 306.151,Z 499.812,A -85,B 0,C 180,E1 -16112.628,E2 -16112.628} C_VEL
LIN {X 0,Y 306.431,Z 498.851,A -85,B 0,C 180,E1 -16113.942,E2 -16113.942} C_VEL
LIN {X 0,Y 306.707,Z 497.513,A -85,B 0,C 180,E1 -16115.256,E2 -16115.256} C_VEL
LIN {X 0,Y 307.015,Z 494.737,A -85,B 0,C 180,E1 -16117.23,E2 -16117.23} C_VEL
LIN {X 0,Y 307.782,Z 490.908,A -85,B 0,C 180,E1 -16119.194,E2 -16119.194} C_VEL
LIN {X 0,Y 308.832,Z 485.927,A -85,B 0,C 180,E1 -16121.15,E2 -16121.15} C_VEL
LIN {X 0,Y 309.778,Z 479.69,A -85,B 0,C 180,E1 -16123.109,E2 -16123.109} C_VEL
LIN {X 0,Y 311.026,Z 471.904,A -85,B 0,C 180,E1 -16125.058,E2 -16125.058} C_VEL
LIN {X 0,Y 312.295,Z 463.916,A -85,B 0,C 180,E1 -16126.671,E2 -16126.671} C_VEL
LIN {X 0,Y 313.449,Z 455.2,A -85,B 0,C 180,E1 -16128.122,E2 -16128.122} C_VEL
LIN {X 0,Y 314.659,Z 444.378,A -85,B 0,C 180,E1 -16129.571,E2 -16129.571} C_VEL
LIN {X 0,Y 315.725,Z 434.068,A -85,B 0,C 180,E1 -16130.662,E2 -16130.662} C_VEL
LIN {X 0,Y 316.667,Z 421.473,A -85,B 0,C 180,E1 -16131.699,E2 -16131.699} C_VEL
LIN {X 0,Y 316.84,Z 415.302,A -85,B 0,C 180,E1 -16132.108,E2 -16132.108} C_VEL
LIN {X 0,Y 313.155,Z 403.051,A -85,B 0,C 180,E1 -16133.052,E2 -16133.052} C_VEL
LIN {X 0,Y 309.817,Z 393.736,A -85,B 0,C 180,E1 -16133.679,E2 -16133.679} C_VEL
LIN {X 0,Y 309.596,Z 384.258,A -85,B 0,C 180,E1 -16137.708,E2 -16137.708} C_VEL
LIN {X 0,Y 309.695,Z 376.051,A -85,B 0,C 180,E1 -16141.458,E2 -16141.458} C_VEL
LIN {X 0,Y 309.934,Z 367.928,A -85,B 0,C 180,E1 -16145.28,E2 -16145.28} C_VEL
LIN {X 0,Y 309.761,Z 363.608,A -85,B 0,C 180,E1 -16147.429,E2 -16147.429} C_VEL
LIN {X 0,Y 308.822,Z 357.795,A -85,B 0,C 180,E1 -16150.381,E2 -16150.381} C_VEL
LIN {X 0,Y 307.716,Z 352.255,A -85,B 0,C 180,E1 -16153.244,E2 -16153.244} C_VEL
LIN {X 0,Y 306.22,Z 345.85,A -85,B 0,C 180,E1 -16156.486,E2 -16156.486} C_VEL
LIN {X 0,Y 305.484,Z 342.745,A -85,B 0,C 180,E1 -16158.07,E2 -16158.07} C_VEL
LIN {X 0,Y 305.505,Z 342.74,A -85,B 0,C 180,E1 -16161.601,E2 -16161.601} C_VEL
LIN {X 0,Y 305.446,Z 342.748,A -85,B 0,C 180,E1 -16164.884,E2 -16164.884} C_VEL
LIN {X 0,Y 305.434,Z 342.753,A -85,B 0,C 180,E1 -16168.352,E2 -16168.352} C_VEL
LIN {X 0,Y 305.501,Z 342.741,A -85,B 0,C 180,E1 -16171.111,E2 -16171.111} C_VEL
LIN {X 0,Y 305.522,Z 342.731,A -85,B 0,C 180,E1 -16173.669,E2 -16173.669} C_VEL
LIN {X 0,Y 304.9,Z 342.817,A -85,B 0,C 180,E1 -16174.769,E2 -16174.769} C_VEL
LIN {X 0,Y 302.018,Z 343.182,A -85,B 0,C 180,E1 -16176.559,E2 -16176.559} C_VEL
LIN {X 0,Y 299.563,Z 343.49,A -85,B 0,C 180,E1 -16178.011,E2 -16178.011} C_VEL
LIN {X 0,Y 298.539,Z 343.613,A -85,B 0,C 180,E1 -16179.137,E2 -16179.137} C_VEL
LIN {X 0,Y 298.474,Z 343.618,A -85,B 0,C 180,E1 -16179.518,E2 -16179.518} C_VEL
LIN {X 0,Y 298.521,Z 343.606,A -85,B 0,C 180,E1 -16182.178,E2 -16182.178} C_VEL
LIN {X 0,Y 298.572,Z 343.595,A -85,B 0,C 180,E1 -16184.993,E2 -16184.993} C_VEL
LIN {X 0,Y 298.574,Z 343.603,A -85,B 0,C 180,E1 -16189.145,E2 -16189.145} C_VEL
LIN {X 0,Y 298.736,Z 343.58,A -85,B 0,C 180,E1 -16191.885,E2 -16191.885} C_VEL
LIN {X 0,Y 298.636,Z 343.589,A -85,B 0,C 180,E1 -16194.598,E2 -16194.598} C_VEL
LIN {X 0,Y 298.899,Z 343.566,A -85,B 0,C 180,E1 -16198.652,E2 -16198.652} C_VEL
LIN {X 0,Y 298.906,Z 343.551,A -85,B 0,C 180,E1 -16201.347,E2 -16201.347} C_VEL
LIN {X 0,Y 298.646,Z 343.597,A -85,B 0,C 180,E1 -16205.401,E2 -16205.401} C_VEL
LIN {X 0,Y 298.736,Z 343.587,A -85,B 0,C 180,E1 -16208.114,E2 -16208.114} C_VEL
LIN {X 0,Y 298.533,Z 343.613,A -85,B 0,C 180,E1 -16212.232,E2 -16212.232} C_VEL
LIN {X 0,Y 298.583,Z 343.605,A -85,B 0,C 180,E1 -16215.21,E2 -16215.21} C_VEL
LIN {X 0,Y 298.543,Z 343.61,A -85,B 0,C 180,E1 -16219.685,E2 -16219.685} C_VEL
LIN {X 0,Y 298.468,Z 343.617,A -85,B 0,C 180,E1 -16223.596,E2 -16223.596} C_VEL
LIN {X 0,Y 298.498,Z 343.703,A -85,B 0,C 180,E1 -16224.888,E2 -16224.888} C_VEL
LIN {X 0,Y 300.751,Z 352.144,A -85,B 0,C 180,E1 -16229.388,E2 -16229.388} C_VEL
LIN {X 0,Y 303.262,Z 361.258,A -85,B 0,C 180,E1 -16233.792,E2 -16233.792} C_VEL
LIN {X 0,Y 305.624,Z 369.724,A -85,B 0,C 180,E1 -16237.544,E2 -16237.544} C_VEL
LIN {X 0,Y 308.083,Z 378.579,A -85,B 0,C 180,E1 -16241.173,E2 -16241.173} C_VEL
LIN {X 0,Y 311.43,Z 390.347,A -85,B 0,C 180,E1 -16245.613,E2 -16245.613} C_VEL
LIN {X 0,Y 314.09,Z 400.487,A -85,B 0,C 180,E1 -16249.122,E2 -16249.122} C_VEL
LIN {X 0,Y 313.675,Z 403.121,A -85,B 0,C 180,E1 -16249.903,E2 -16249.903} C_VEL
LIN {X 0,Y 311.058,Z 412.641,A -85,B 0,C 180,E1 -16252.572,E2 -16252.572} C_VEL
LIN {X 0,Y 314.222,Z 436.086,A -85,B 0,C 180,E1 -16253.761,E2 -16253.761} C_VEL
LIN {X 0,Y 316.54,Z 453.741,A -85,B 0,C 180,E1 -16254.928,E2 -16254.928} C_VEL
LIN {X 0,Y 318.028,Z 469.932,A -85,B 0,C 180,E1 -16256.206,E2 -16256.206} C_VEL
LIN {X 0,Y 315.897,Z 484.432,A -85,B 0,C 180,E1 -16257.354,E2 -16257.354} C_VEL
LIN {X 0,Y 313.439,Z 498.57,A -85,B 0,C 180,E1 -16258.72,E2 -16258.72} C_VEL
LIN {X 0,Y 310.631,Z 513.806,A -85,B 0,C 180,E1 -16260.526,E2 -16260.526} C_VEL
LIN {X 0,Y 307.863,Z 527.318,A -85,B 0,C 180,E1 -16262.47,E2 -16262.47} C_VEL
LIN {X 0,Y 305.467,Z 538.819,A -85,B 0,C 180,E1 -16264.448,E2 -16264.448} C_VEL
LIN {X 0,Y 303.132,Z 550.308,A -85,B 0,C 180,E1 -16266.792,E2 -16266.792} C_VEL
LIN {X 0,Y 301.333,Z 559.596,A -85,B 0,C 180,E1 -16269.033,E2 -16269.033} C_VEL
LIN {X 0,Y 299.826,Z 568.44,A -85,B 0,C 180,E1 -16271.556,E2 -16271.556} C_VEL
LIN {X 0,Y 298.575,Z 576.534,A -85,B 0,C 180,E1 -16274.368,E2 -16274.368} C_VEL
LIN {X 0,Y 297.882,Z 582.797,A -85,B 0,C 180,E1 -16277.052,E2 -16277.052} C_VEL
LIN {X 0,Y 297.529,Z 587.932,A -85,B 0,C 180,E1 -16279.799,E2 -16279.799} C_VEL
LIN {X 0,Y 297.482,Z 592.199,A -85,B 0,C 180,E1 -16282.857,E2 -16282.857} C_VEL
LIN {X 0,Y 297.638,Z 595.006,A -85,B 0,C 180,E1 -16285.941,E2 -16285.941} C_VEL
LIN {X 0,Y 297.615,Z 596.156,A -85,B 0,C 180,E1 -16288.65,E2 -16288.65} C_VEL
LIN {X 0,Y 297.596,Z 596.233,A -85,B 0,C 180,E1 -16291.356,E2 -16291.356} C_VEL
LIN {X 0,Y 297.653,Z 595.176,A -85,B 0,C 180,E1 -16294.065,E2 -16294.065} C_VEL
LIN {X 0,Y 297.457,Z 592.631,A -85,B 0,C 180,E1 -16297.105,E2 -16297.105} C_VEL
LIN {X 0,Y 297.403,Z 588.655,A -85,B 0,C 180,E1 -16300.212,E2 -16300.212} C_VEL
LIN {X 0,Y 297.785,Z 583.982,A -85,B 0,C 180,E1 -16302.959,E2 -16302.959} C_VEL
LIN {X 0,Y 298.528,Z 578.09,A -85,B 0,C 180,E1 -16305.711,E2 -16305.711} C_VEL
LIN {X 0,Y 299.746,Z 571.043,A -85,B 0,C 180,E1 -16308.456,E2 -16308.456} C_VEL
LIN {X 0,Y 301.566,Z 562.165,A -85,B 0,C 180,E1 -16311.347,E2 -16311.347} C_VEL
LIN {X 0,Y 304.145,Z 551.592,A -85,B 0,C 180,E1 -16314.218,E2 -16314.218} C_VEL
LIN {X 0,Y 307.43,Z 539.638,A -85,B 0,C 180,E1 -16316.931,E2 -16316.931} C_VEL
LIN {X 0,Y 311.1,Z 526.56,A -85,B 0,C 180,E1 -16319.432,E2 -16319.432} C_VEL
LIN {X 0,Y 315.45,Z 511.877,A -85,B 0,C 180,E1 -16321.762,E2 -16321.762} C_VEL
LIN {X 0,Y 319.689,Z 497.109,A -85,B 0,C 180,E1 -16323.72,E2 -16323.72} C_VEL
LIN {X 0,Y 324.159,Z 481.219,A -85,B 0,C 180,E1 -16325.45,E2 -16325.45} C_VEL
LIN {X 0,Y 325.869,Z 474.427,A -85,B 0,C 180,E1 -16326.118,E2 -16326.118} C_VEL
LIN {X 0,Y 327.213,Z 462.002,A -85,B 0,C 180,E1 -16327.518,E2 -16327.518} C_VEL
LIN {X 0,Y 328.585,Z 448.334,A -85,B 0,C 180,E1 -16328.965,E2 -16328.965} C_VEL
LIN {X 0,Y 328.648,Z 436.134,A -85,B 0,C 180,E1 -16330.44,E2 -16330.44} C_VEL
LIN {X 0,Y 328.327,Z 427.855,A -85,B 0,C 180,E1 -16331.576,E2 -16331.576} C_VEL
LIN {X 0,Y 327.907,Z 422.19,A -85,B 0,C 180,E1 -16332.472,E2 -16332.472} C_VEL
LIN {X 0,Y 326.407,Z 418.57,A -85,B 0,C 180,E1 -16333.589,E2 -16333.589} C_VEL
LIN {X 0,Y 324.653,Z 415.531,A -85,B 0,C 180,E1 -16334.992,E2 -16334.992} C_VEL
LIN {X 0,Y 323.622,Z 413.973,A -85,B 0,C 180,E1 -16335.979,E2 -16335.979} C_VEL
LIN {X 0,Y 322.305,Z 411.719,A -85,B 0,C 180,E1 -16337.853,E2 -16337.853} C_VEL
LIN {X 0,Y 321.601,Z 410.673,A -85,B 0,C 180,E1 -16339.898,E2 -16339.898} C_VEL
LIN {X 0,Y 321.863,Z 410.815,A -85,B 0,C 180,E1 -16342.31,E2 -16342.31} C_VEL
LIN {X 0,Y 322.661,Z 413.799,A -85,B 0,C 180,E1 -16344.734,E2 -16344.734} C_VEL
LIN {X 0,Y 323.513,Z 416.989,A -85,B 0,C 180,E1 -16346.37,E2 -16346.37} C_VEL
LIN {X 0,Y 325.241,Z 422.991,A -85,B 0,C 180,E1 -16348.762,E2 -16348.762} C_VEL
LIN {X 0,Y 326.734,Z 428.797,A -85,B 0,C 180,E1 -16350.633,E2 -16350.633} C_VEL
LIN {X 0,Y 327.957,Z 434.985,A -85,B 0,C 180,E1 -16352.302,E2 -16352.302} C_VEL
LIN {X 0,Y 328.468,Z 439.157,A -85,B 0,C 180,E1 -16353.3,E2 -16353.3} C_VEL
LIN {X 0,Y 326.902,Z 444.607,A -85,B 0,C 180,E1 -16354.022,E2 -16354.022} C_VEL
LIN {X 0,Y 323.226,Z 455.802,A -85,B 0,C 180,E1 -16355.599,E2 -16355.599} C_VEL
LIN {X 0,Y 318.949,Z 468.243,A -85,B 0,C 180,E1 -16357.78,E2 -16357.78} C_VEL
LIN {X 0,Y 315.206,Z 478.445,A -85,B 0,C 180,E1 -16359.979,E2 -16359.979} C_VEL
LIN {X 0,Y 311.442,Z 488.085,A -85,B 0,C 180,E1 -16362.603,E2 -16362.603} C_VEL
LIN {X 0,Y 308.742,Z 494.465,A -85,B 0,C 180,E1 -16364.825,E2 -16364.825} C_VEL
LIN {X 0,Y 306.693,Z 498.899,A -85,B 0,C 180,E1 -16366.753,E2 -16366.753} C_VEL
LIN {X 0,Y 304.38,Z 503.324,A -85,B 0,C 180,E1 -16369.356,E2 -16369.356} C_VEL
LIN {X 0,Y 302.652,Z 506.128,A -85,B 0,C 180,E1 -16371.992,E2 -16371.992} C_VEL
LIN {X 0,Y 301.392,Z 507.419,A -85,B 0,C 180,E1 -16374.649,E2 -16374.649} C_VEL
LIN {X 0,Y 300.855,Z 507.484,A -85,B 0,C 180,E1 -16375.982,E2 -16375.982} C_VEL
LIN {X 0,Y 299.95,Z 506.417,A -85,B 0,C 180,E1 -16378.658,E2 -16378.658} C_VEL
LIN {X 0,Y 299.626,Z 505.288,A -85,B 0,C 180,E1 -16380.001,E2 -16380.001} C_VEL
LIN {X 0,Y 299.496,Z 503.74,A -85,B 0,C 180,E1 -16381.345,E2 -16381.345} C_VEL
LIN {X 0,Y 299.379,Z 500.626,A -85,B 0,C 180,E1 -16383.365,E2 -16383.365} C_VEL
LIN {X 0,Y 299.37,Z 496.543,A -85,B 0,C 180,E1 -16385.389,E2 -16385.389} C_VEL
LIN {X 0,Y 299.597,Z 491.407,A -85,B 0,C 180,E1 -16387.414,E2 -16387.414} C_VEL
LIN {X 0,Y 300.214,Z 485.103,A -85,B 0,C 180,E1 -16389.432,E2 -16389.432} C_VEL
LIN {X 0,Y 300.893,Z 476.164,A -85,B 0,C 180,E1 -16391.793,E2 -16391.793} C_VEL
LIN {X 0,Y 301.777,Z 466.835,A -85,B 0,C 180,E1 -16393.811,E2 -16393.811} C_VEL
LIN {X 0,Y 302.786,Z 455.585,A -85,B 0,C 180,E1 -16395.827,E2 -16395.827} C_VEL
LIN {X 0,Y 304.008,Z 444.438,A -85,B 0,C 180,E1 -16397.49,E2 -16397.49} C_VEL
LIN {X 0,Y 305.206,Z 431.283,A -85,B 0,C 180,E1 -16399.128,E2 -16399.128} C_VEL
LIN {X 0,Y 306.373,Z 418.092,A -85,B 0,C 180,E1 -16400.477,E2 -16400.477} C_VEL
LIN {X 0,Y 307.061,Z 409.553,A -85,B 0,C 180,E1 -16401.218,E2 -16401.218} C_VEL
LIN {X 0,Y 303.875,Z 394.375,A -85,B 0,C 180,E1 -16402.572,E2 -16402.572} C_VEL
LIN {X 0,Y 300.21,Z 379.095,A -85,B 0,C 180,E1 -16403.709,E2 -16403.709} C_VEL
LIN {X 0,Y 298.966,Z 374.114,A -85,B 0,C 180,E1 -16404.061,E2 -16404.061} C_VEL
LIN {X 0,Y 299.385,Z 367.876,A -85,B 0,C 180,E1 -16408.002,E2 -16408.002} C_VEL
LIN {X 0,Y 299.819,Z 362.124,A -85,B 0,C 180,E1 -16411.757,E2 -16411.757} C_VEL
LIN {X 0,Y 300.17,Z 357.335,A -85,B 0,C 180,E1 -16414.964,E2 -16414.964} C_VEL
LIN {X 0,Y 300.073,Z 353.687,A -85,B 0,C 180,E1 -16417.514,E2 -16417.514} C_VEL
LIN {X 0,Y 299.369,Z 348.803,A -85,B 0,C 180,E1 -16421.097,E2 -16421.097} C_VEL
LIN {X 0,Y 299.028,Z 346.82,A -85,B 0,C 180,E1 -16422.743,E2 -16422.743} C_VEL
LIN {X 0,Y 300.398,Z 351.827,A -85,B 0,C 180,E1 -16425.42,E2 -16425.42} C_VEL
LIN {X 0,Y 301.779,Z 358.261,A -85,B 0,C 180,E1 -16428.774,E2 -16428.774} C_VEL
LIN {X 0,Y 302.899,Z 364.663,A -85,B 0,C 180,E1 -16432.082,E2 -16432.082} C_VEL
LIN {X 0,Y 303.164,Z 369.017,A -85,B 0,C 180,E1 -16434.232,E2 -16434.232} C_VEL
LIN {X 0,Y 302.953,Z 376.38,A -85,B 0,C 180,E1 -16437.751,E2 -16437.751} C_VEL
LIN {X 0,Y 302.862,Z 386.447,A -85,B 0,C 180,E1 -16442.345,E2 -16442.345} C_VEL
LIN {X 0,Y 303.027,Z 394.77,A -85,B 0,C 180,E1 -16445.894,E2 -16445.894} C_VEL
LIN {X 0,Y 307.882,Z 408.568,A -85,B 0,C 180,E1 -16446.857,E2 -16446.857} C_VEL
LIN {X 0,Y 310.375,Z 417.753,A -85,B 0,C 180,E1 -16447.611,E2 -16447.611} C_VEL
LIN {X 0,Y 309.571,Z 429.64,A -85,B 0,C 180,E1 -16448.489,E2 -16448.489} C_VEL
LIN {X 0,Y 308.567,Z 441.337,A -85,B 0,C 180,E1 -16449.635,E2 -16449.635} C_VEL
LIN {X 0,Y 307.354,Z 452.12,A -85,B 0,C 180,E1 -16450.98,E2 -16450.98} C_VEL
LIN {X 0,Y 306.081,Z 460.661,A -85,B 0,C 180,E1 -16452.285,E2 -16452.285} C_VEL
LIN {X 0,Y 304.83,Z 469.408,A -85,B 0,C 180,E1 -16453.936,E2 -16453.936} C_VEL
LIN {X 0,Y 303.401,Z 477.934,A -85,B 0,C 180,E1 -16455.92,E2 -16455.92} C_VEL
LIN {X 0,Y 302.342,Z 484.736,A -85,B 0,C 180,E1 -16457.921,E2 -16457.921} C_VEL
LIN {X 0,Y 301.253,Z 490.163,A -85,B 0,C 180,E1 -16459.92,E2 -16459.92} C_VEL
LIN {X 0,Y 300.198,Z 494.444,A -85,B 0,C 180,E1 -16461.922,E2 -16461.922} C_VEL
LIN {X 0,Y 299.842,Z 496.663,A -85,B 0,C 180,E1 -16463.267,E2 -16463.267} C_VEL
